// TwinCAT 3 PLC project CX747246
// ProgramVersion: 3.1.4024.0
// libraries:
//   CmpBitmapPool, * (System)
//   Tc2_Standard, * (Beckhoff Automation GmbH)
//   Tc2_SUPS, * (Beckhoff Automation GmbH)
//   Tc2_System, * (Beckhoff Automation GmbH)
//   Tc2_Utilities, * (Beckhoff Automation GmbH)
//   Tc3_EventLogger, * (Beckhoff Automation GmbH)
//   Tc3_Module, * (Beckhoff Automation GmbH)
//   VisuDialogs, * (System)
//   VisuElemEventTable, * (System)
//   VisuUserMgmt, * (System)
//   Visu Utils,3.5.12.0,System
//   VisuSymbols,3.5.10.0,System
// project tree:
//   DUTs/ StrFuncParoEnviar.TcDUT, Str_Config_ADS_to_PLC.TcDUT, Str_HistTablasMySQL.TcDUT
//   / GlobalTextList.TcGTLO, Lectura_PLCs_1.TcTTO, PlcTask.TcTTO, VISU_TASK.TcTTO
//   GVLs/ Fecha_PLC.TcGVL, Lectura_PLCs.TcGVL, RegistroLocalDataBase.TcGVL, Var_Com_CH4_MulDis.TcGVL
//   POUs/Events_Alarms/ Eventos_PLC.TcPOU, Events.TcPOU
//   POUs/FBs/ fbLectura_a_PLC.TcPOU, fb_Funciones_Paro.TcPOU, FuncGeneralesCortHum4.TcPOU, FuncGeneralesMult1.TcPOU, FuncGeneralesMult2.TcPOU, TempParoAcumulad.TcPOU
//   POUs/Funciones comunes/ Fecha_Hora_PLC.TcPOU, HMI.TcPOU, Utilidades.TcPOU
//   POUs/Lectura_a_PLC_Maestro/ Lectura_Maestro.TcPOU, MAIN_Orden_Lectura_PLCs.TcPOU
//   POUs/ MAIN.TcPOU
//   POUs/PRGs_Nodos/ FuncParoNodoMultidiscos.TcPOU, FuncParoNodoCorteH4Remote1.TcPOU
//   VISUs/ Ajustes_Multidiscos1.TcVIS, Ajustes_Multidiscos2.TcVIS, DiagnosticoFB.TcVIS, Home_CortH4.TcVIS, Home_Multidis1.TcVIS, Home_Multidis2.TcVIS, ImagePool.TcIPO (not stored), Modelo_Tabla_Ch4.TcVIS, Ajustes_CorteH4.TcVIS, Home_Sel_Maq.TcVIS, HistTablaTablas_Ch4.TcVIS, Modelo_Tabla_Md1.TcVIS, Modelo_Tabla_Md2.TcVIS, VisualizationManager.TcVMO (not stored), V_Emerg_Fin_Prod_Ch4.TcVIS, V_Emerg_Fin_Prod_Md2.TcVIS, V_Emerg_Fin_Prod_Md1.TcVIS
//   VISUs/IMAGENES/ Imagenes.TcIPO (not stored)
//   VISUs/Listas_Para_Desplegables/ FormatoTabla.TcTLO
// real-time tasks:
//   TASK PlcTask: cycle T#10ms, priority 20, ADS port 350
//   TASK VISU_TASK: cycle T#200000us, priority 30, ADS port 352
//   TASK Lectura_PLCs: cycle T#10ms, priority 1, ADS port 351
// I/O:
//   DEVICE Device 2 (EtherCAT), AmsNetId 5.116.114.70.3.1
//     Term 1 (EK1200) [EK1200-5000 EtherCAT Power supply (2A E-Bus)]
//       Term 2 (EL1859) [EL1859 8Ch. Dig. Input 24V, 3ms, 8Ch. Dig. Output 24V, 0.5A]
//       Term 3 (EK1110) [EK1110 EtherCAT extension]
//     Term 4 (EK1100) [EK1100 EtherCAT Coupler (2A E-Bus)]
//       Term 5 (EL1859) [EL1859 8Ch. Dig. Input 24V, 3ms, 8Ch. Dig. Output 24V, 0.5A]
//       Term 6 (EL9011) [EL9011 End Terminal]
// variable links:
//   CX747246/CX747246 Instance <-> Device 2 (EtherCAT)/Term 1 (EK1200)/Term 2 (EL1859)
//     PlcTask Inputs/MAIN.id0Local <-> Channel 1/Input
//     PlcTask Inputs/MAIN.id0Local @bit {1..7} <-> Channel {2..8}/Input  (7 links)
//     PlcTask Outputs/MAIN.od0Local @bit {1..7} <-> Channel {10..16}/Output  (7 links)
//     PlcTask Outputs/MAIN.od0Local <-> Channel 9/Output
//   CX747246/CX747246 Instance <-> Device 2 (EtherCAT)/Term 4 (EK1100)/Term 5 (EL1859)
//     PlcTask Inputs/MAIN.id0Remoto1 <-> Channel 1/Input
//     PlcTask Inputs/MAIN.id0Remoto1 @bit {1..7} <-> Channel {2..8}/Input  (7 links)
//     PlcTask Outputs/MAIN.od0Remoto1 @bit {1..7} <-> Channel {10..16}/Output  (7 links)
//     PlcTask Outputs/MAIN.od0Remoto1 <-> Channel 9/Output

CONFIGURATION CX747246
    RESOURCE PLC ON TwinCAT3
        TASK Lectura_PLCs_1(INTERVAL := T#10ms, PRIORITY := 1);
        TASK PlcTask(INTERVAL := T#10ms, PRIORITY := 20);
        TASK VISU_TASK(INTERVAL := T#200000us, PRIORITY := 30);
        PROGRAM MAIN_Orden_Lectura_PLCs WITH Lectura_PLCs_1 : MAIN_Orden_Lectura_PLCs;
        PROGRAM MAIN WITH PlcTask : MAIN;
        PROGRAM VisuElems_Visu_Prg WITH VISU_TASK : VisuElems.Visu_Prg;
        PROGRAM HMI WITH VISU_TASK : HMI;
    END_RESOURCE
END_CONFIGURATION

// ---- DUTs/StrFuncParoEnviar.TcDUT
TYPE StrFuncParoEnviar :
STRUCT
	Cont_Piezas:INT;//Numero de piezas actuales
	Min_Parado_Ftc:INT;//Minutos actuales parado
	t_Entr_Piez_Ante_Ftc:TIME;//Tiempo entre piezas tabla anterior
	t_Entre_Piez_Ftc:TIME;//Tiempo actual entre piezas
	H_InParo_Ftc:STRING;//Variable de la hora de inicio del paro tipo STRING
	H_FinParo_Ftc:STRING;//Hora Fin del paro
	S_Justi_Paro_Ftc:STRING;//Justificación del paro string
	Fotocelula:BOOL;//Fotocelula física
	MParo_Ftc:BOOL;//Marca de paro 
	M_SinParo_Ftc:BOOL;//Marca de sin paro activo
	tFiltro_up_Ftc:BOOL;//Q del temporizador Up filtro fotocelula 
	tFiltro_down_Ftc:BOOL;//Q del temporizador Down filtro fotocelula 	
END_STRUCT
END_TYPE

// ---- DUTs/Str_Config_ADS_to_PLC.TcDUT
TYPE Str_Config_ADS_to_PLC :
STRUCT
    NETID     : T_AmsNetId;
    PORT      : T_AmsPort;
    IDXGRP    : UDINT;
    IDXOFFS   : UDINT;
    LEN       : UDINT;
    DESTADDR  : PVOID;
    READ      : BOOL;
    TMOUT     : TIME := DEFAULT_ADS_TIMEOUT;
	
//Output
	BUSY    : BOOL;
    ERR     : BOOL;
    ERRID   : UDINT;
END_STRUCT
END_TYPE

// ---- DUTs/Str_HistTablasMySQL.TcDUT
TYPE Str_HistTablasMySQL :
STRUCT
	ID:INT;
	Fecha:STRING;
	Modelo:STRING;
	Formato:STRING;
	Espesor:STRING;
	Maquina :STRING;	
	Cont_Piezas:INT;//Numero de piezas actuales
	t_Entre_Piez_Ftc:TIME;//Tiempo actual entre piezas
	S_Justi_Paro_Ftc:STRING;//Justificación del paro string	
END_STRUCT
END_TYPE

// ---- GVLs/Fecha_PLC.TcGVL
{attribute 'qualified_only'}
VAR_GLOBAL
	fbGetLocalSystemTime:FB_LocalSystemTime; //Lee la hora local del PLC 
	Fecha_Segundos:DINT;
	StringDateTime:STRING;
	StringDateHourMin:STRING;
	StringDate:STRING;
	StringTime:STRING;
	StringHora:STRING;
	StringMinutos:STRING;
	StringSegundos:STRING;
	StringMes:STRING;
	StringDia:STRING;
	StringAno:STRING;
	
	//concatenaciones de strings
	Mes_Dia_Hora_Min_Real:STRING;
	//Tipo time para poder restar horas 
	Fecha_Entera_Dt:DT;	
	Fecha_Struct: Tc2_Utilities.TIMESTRUCT;
	Fecha_Time_PLC:TIME;
	
END_VAR

// ---- GVLs/Lectura_PLCs.TcGVL
{attribute 'qualified_only'}
VAR_GLOBAL
										//	Variables Lectura de PLC Maestro
									
//Las marcas a las que hace referencia del plc Maestro para las Bool van de la %MB46110 a %MB46210
	aMasterBoolCom:ARRAY[0..100] OF BOOL;
	
//Las marcas a las que hace referencia del plc Maestro para las string van de la %MW41300 a %MW42515   
	aMasterStringCom:ARRAY[0..14] OF STRING;
	
//Las marcas a las que hace rreferencia del plc Maestro para las Time van de la %MW47210 a %MW47414
	aMasterTimeCom:ARRAY[0..50]OF TIME;	
	
//Las marcas a las que hace referencia del plc Maestro para las Words van de la %MW45050 a %MW45090
	aMasterWordCom:ARRAY[0..40] OF WORD;	

END_VAR

// ---- GVLs/RegistroLocalDataBase.TcGVL
{attribute 'qualified_only'}
VAR_GLOBAL
	aValoresTurnosAnt: ARRAY [0..50] OF StrFuncParoEnviar;//Cada fin de turno se envía los valores de la ultima tabla que ha psado y se queda guardado en esta array para enseñarlo por el Scada
END_VAR
VAR_GLOBAL PERSISTENT
	//Array para el histórico de las tablas enviado a la base de datos
	 aHistoricStrTablasCH4: ARRAY[0..100]OF Str_HistTablasMySQL;
	 aHistoricStrTablasMD1: ARRAY[0..100]OF Str_HistTablasMySQL;
	 aHistoricStrTablasMD2: ARRAY[0..100]OF Str_HistTablasMySQL;
END_VAR

// ---- GVLs/Var_Com_CH4_MulDis.TcGVL
{attribute 'qualified_only'}
VAR_GLOBAL
	// Variables Escritura en PLC Maestro 
	aStringCom AT %MW2000: ARRAY[0..97] OF STRING;	//(1 string = 81 MW)
	aWordCom AT %MW10000: ARRAY[0..249] OF WORD;	//(1 Word = 1MW)
	aBoolCom AT %MB10250: ARRAY[0..499] OF BOOL;	//(1 Bool = 1MB)
	aTimeCom AT %MW10750: ARRAY[0..124] OF TIME;	//(1 Time = 4MW)
END_VAR

// ---- POUs/Lectura_a_PLC_Maestro/MAIN_Orden_Lectura_PLCs.TcPOU
PROGRAM MAIN_Orden_Lectura_PLCs
VAR
	bHabilitarLecturaDePLCs : BOOL := TRUE;
	bHabilitaLectura_Maestro : BOOL:=TRUE;
	State_Lectura_PLC: (READING_PLC_WAITING, READING_PLC_MAESTRO, FINISH_ALL_OK);
	tReadState_Entre_Lecturas_PLCs:ton:=(PT:=T#5MS);
END_VAR

// POU para ordenar la lectura de los distintos PLCs para que nunca lean a la vez 

CASE State_Lectura_PLC OF 

	READING_PLC_WAITING:tReadState_Entre_Lecturas_PLCs(IN:=FALSE);	

	READING_PLC_MAESTRO:	IF bHabilitaLectura_Maestro THEN
						tReadState_Entre_Lecturas_PLCs(IN:=TRUE);	
							IF tReadState_Entre_Lecturas_PLCs.Q THEN 
								tReadState_Entre_Lecturas_PLCs(IN:=FALSE);
								Lectura_Maestro();
								Lectura_Maestro.fbLectura_a_PLC_Maestro.SetStartReading();
							END_IF
							IF Lectura_Maestro.bNextBlockToRead_L4_Done THEN

								Lectura_Maestro.fbLectura_a_PLC_Maestro.SetFalseBlockReadDone();
								State_Lectura_PLC := FINISH_ALL_OK; //Cuando se añada un PLC cambiad el nombre.
							END_IF
						ELSE 
							State_Lectura_PLC := FINISH_ALL_OK; //Cuando se añada un PLC cambiad el nombre.
							Lectura_Maestro.fbLectura_a_PLC_Maestro.SetFalseBlockReadDone();
					END_IF
					
	FINISH_ALL_OK: tReadState_Entre_Lecturas_PLCs(IN:=FALSE);	
					State_Lectura_PLC := READING_PLC_Maestro;				

END_CASE



//Habilitar la lectura de los PLCs
IF bHabilitarLecturaDePLCs THEN 
	SetStartReadingPLCs();
	ELSE
		State_Lectura_PLC:=READING_PLC_WAITING;
END_IF

METHOD SetStartReadingPLCs : BOOL
VAR_INPUT
END_VAR
IF State_Lectura_PLC = READING_PLC_WAITING THEN 
	State_Lectura_PLC := READING_PLC_Maestro;
END_IF
END_METHOD

END_PROGRAM

// ---- POUs/Lectura_a_PLC_Maestro/Lectura_Maestro.TcPOU
PROGRAM Lectura_Maestro
VAR
	// >>>>>>>>>>>>>>>>>>>>>>>>>>>>>>>>>>>>>>>>   Estructuras de configuración con la comunicación desde y hacia el PLC Maestro <<<<<<<<<<<<<<<<<<<<<<<<<<<<<<<<<<<<<<<<<<<<<<<<<
	
	//Recordar que el IDXOFFS debe ser el doble de la posición a la que queréis acceder Ejemplo: para leer los strings a partir de la dirección MW100 Debéis poner 200 en exadecimal (C8)
	
	//Configuración de la lectura de las variables Bool, IDXGRP:=16#4020(Hace referencia a la lectura de M),IDXOFFS:=16#B41E(%MB46110 a %MB46210), LEN : 101 Longitud bools leidos,DESTADDR:= ADR(Lectura_PLCs.aMasterBoolCom) Ubicación del array donde se guarda la lectura
	Config_Read_ADS_Bools_Maestro:Str_Config_ADS_to_PLC:=(NETID:='192.168.10.71.1.1', PORT:=851, IDXGRP:=16#4020,IDXOFFS:=16#B41E,LEN:=101,DESTADDR:= ADR(Lectura_PLCs.aMasterBoolCom));
	
	//Configuración de la lectura de las variables String, IDXGRP:=16#4020(Hace referencia a la lectura de M),IDXOFFS:= 16#142A8(%MW41300 a %MW42515 ( 15 word)),Longitud de bytes a leer 1215 bytes = 15 strings que son 81words por cada string. ,DESTADDR:= ADR(Lectura_PLCs.aMasterStringCom) Ubicación del array donde se guarda la lectura
	Config_Read_ADS_Strings_Maestro:Str_Config_ADS_to_PLC:=(NETID:='192.168.10.71.1.1', PORT:=851, IDXGRP:=16#4020,IDXOFFS:=16#142A8,LEN:=1215,DESTADDR:= ADR(Lectura_PLCs.aMasterStringCom));
	
	//Configuración de la lectura de las variables Times, IDXGRP:=16#4020(Hace referencia a la lectura de M),IDXOFFS:=16#16F30 ( %MW47210 a %MW47414 (204 word),LEN:= 204 Longitud de bytes a leer bytes = 200words    51 componentes,DESTADDR:= ADR(Lectura_PLCs.aMasterTimeCom) Ubicación del array donde se guarda la lectura
	Config_Read_ADS_Times_Maestro:Str_Config_ADS_to_PLC:=(NETID:='192.168.10.71.1.1', PORT:=851, IDXGRP:=16#4020,IDXOFFS:=16#16F30,LEN:= 204,DESTADDR:= ADR(Lectura_PLCs.aMasterTimeCom));
	
	//Configuración de la lectura de las variables Words, IDXGRP:=16#4020(Hace referencia a la lectura de M),IDXOFFS:=16#15FF4 ( %MW45050 a %MW45090 (40 word),82;//Longitud de bytes a leer 80 bytes = 40words   ,DESTADDR:= ADR(Lectura_PLCs.aMasteWordCom) Ubicación del array donde se guarda la lectura
	Config_Read_ADS_Words_Maestro:Str_Config_ADS_to_PLC:=(NETID:='192.168.10.71.1.1', PORT:=851, IDXGRP:=16#4020,IDXOFFS:=16#15FF4,LEN:=82,DESTADDR:= ADR(Lectura_PLCs.aMasterWordCom));
	
	
	fbLectura_a_PLC_Maestro:fbLectura_a_PLC;
	

END_VAR
VAR_INPUT
	bNextBlockToRead_L4_Done:BOOL;
END_VAR

fbLectura_a_PLC_Maestro(
	Config_PLC_ADS_Bools:=Config_Read_ADS_Bools_Maestro,
	Config_PLC_ADS_Strings:=Config_Read_ADS_Strings_Maestro,
	Config_PLC_ADS_Times:=Config_Read_ADS_Times_Maestro,
	Config_PLC_ADS_Words:=Config_Read_ADS_Words_Maestro,
 	TimeReadStateEntreLecturas:=T#20MS,
	bHabilitadaLectura:=TRUE,
	);

END_PROGRAM

// ---- POUs/FBs/fbLectura_a_PLC.TcPOU
FUNCTION_BLOCK fbLectura_a_PLC
VAR_INPUT
	TimeReadStateEntreLecturas:TIME;
	//Estructuras para la configuración de la lectura de lsa ubicaciones de las variables y los tipos en el PLC 
	Config_PLC_ADS_Bools:Str_Config_ADS_to_PLC;
	Config_PLC_ADS_Strings:Str_Config_ADS_to_PLC;
	Config_PLC_ADS_Times:Str_Config_ADS_to_PLC;
	Config_PLC_ADS_Words:Str_Config_ADS_to_PLC;
	bHabilitadaLectura:BOOL;	
END_VAR 

VAR_OUTPUT
	AlarmaFalloComunicacion:BOOL;
END_VAR
VAR


	
	//Tiempos para el control de las lecturas de los diferentes tipos de variables
	tReadState_Entre_Lecturas:ton;
	eReadState : (EN_ESPERA,READING_BOOLS,READING_STRINGS,READING_TIMES,READING_WORDS,END_ALL_OK);
	//Bits de activación de lectura de las variables
	Execute_Read_Bools:BOOL;
	Execute_Read_Strings:BOOL;
	Execute_Read_Times:BOOL;
	Execute_Read_Words:BOOL;
	
	//Alarmas Errores en las lecturas al PLC 
	Err_fbLecturaBools: BOOL;
	Err_ID_fbLecturaBools: UDINT;
	Err_fbLecturaStrings: BOOL;
	Err_ID_fbLecturaStrings: UDINT;
	Err_fbLecturaTimes: BOOL;
	Err_ID_fbLecturaTimes: UDINT;
	Err_fbLecturaWords: BOOL;
	Err_ID_fbLecturaWords: UDINT;
	
	
	//Instancias de las funciones de lectura
	fbLecturaWords:        adsRead;	
	fbLecturaTimes:        adsRead;	
	fbLecturaStrings:      adsRead;
	fbLecturaBools:        adsRead;
	bBlock_Read_Done : BOOL;
		//Comprobaciones 
	Cont_Bool:INT;
	Cont_Str:INT;
	Cont_Word:INT;
	Cont_Time:INT;
	
	fptReadState_Entre_Lecturas:R_trig;

END_VAR
VAR PERSISTENT

END_VAR

tReadState_Entre_Lecturas(PT:=TimeReadStateEntreLecturas);
CASE eReadState OF 
	EN_ESPERA :   	tReadState_Entre_Lecturas(IN:=FALSE);

	READING_BOOLS : tReadState_Entre_Lecturas(IN:=TRUE);
					Read_Bools();
					IF tReadState_Entre_Lecturas.Q THEN
						tReadState_Entre_Lecturas(IN:=FALSE);
					    Cont_Bool:=Cont_Bool + 1;
						Execute_Read_Bools:=TRUE;
 						eReadState := READING_STRINGS;
					END_IF
	
	READING_STRINGS :tReadState_Entre_Lecturas(IN:=TRUE);
						Read_Strings();
					IF tReadState_Entre_Lecturas.Q THEN 
					    tReadState_Entre_Lecturas(IN:=FALSE);
						Execute_Read_Strings:=TRUE;
						Cont_Str:=Cont_Str + 1;	
						eReadState := READING_TIMES;
			
					END_IF
					
	READING_TIMES : tReadState_Entre_Lecturas(IN:=TRUE);
					Read_Times();
					IF tReadState_Entre_Lecturas.Q THEN 
						tReadState_Entre_Lecturas(IN:=FALSE);
						Execute_Read_Times:=TRUE;
						Cont_Time:=Cont_Time + 1;	
						eReadState := READING_WORDS;	
					END_IF
					
	READING_WORDS : tReadState_Entre_Lecturas(IN:=TRUE);
					Read_Words();
					IF tReadState_Entre_Lecturas.Q THEN 
						tReadState_Entre_Lecturas(IN:=FALSE);
						Execute_Read_Words:=TRUE;
						Cont_Word:=Cont_Word + 1;	
						eReadState := END_ALL_OK;	
									
					END_IF

	END_ALL_OK :// eReadState := READING_BOOLS;
				bBlock_Read_Done:=TRUE;
END_CASE

//En espera en caso de estar deshabilitado
IF NOT bHabilitadaLectura THEN
		eReadState:= EN_ESPERA;
END_IF
IF Err_fbLecturaBools OR Err_fbLecturaStrings OR Err_fbLecturaTimes OR Err_fbLecturaWords THEN 
	AlarmaFalloComunicacion:=TRUE;
	ELSE 
		AlarmaFalloComunicacion:=false;
END_IF

METHOD Read_Bools : BOOL
VAR_INPUT
END_VAR
fbLecturaBools.NETID:=  Config_PLC_ADS_Bools.NETID;//Lee del equipo remoto los Bool 
fbLecturaBools.PORT:=   Config_PLC_ADS_Bools.PORT;
fbLecturaBools.IDXGRP:= Config_PLC_ADS_Bools.IDXGRP;//Variables %M
fbLecturaBools.IDXOFFS:= Config_PLC_ADS_Bools.IDXOFFS;//Offset de la marca que empieza a leer
fbLecturaBools.LEN:= Config_PLC_ADS_Bools.LEN;//Longitud de bits a leer
fbLecturaBools.DESTADDR:= Config_PLC_ADS_Bools.DESTADDR;//Numero componentes
fbLecturaBools.READ:=     Execute_Read_Bools;//Bit de ejecutar la lectura 
fbLecturaBools();
Err_fbLecturaBools := fbLecturaBools.ERR;
Err_ID_fbLecturaBools := fbLecturaBools.ERRID;

Execute_Read_Bools := FALSE;
END_METHOD

METHOD Read_Strings : BOOL
VAR_INPUT
END_VAR
fbLecturaStrings.NETID:=  Config_PLC_ADS_Strings.NETID;//Lee del equipo remoto String
fbLecturaStrings.PORT:=   Config_PLC_ADS_Strings.PORT;
fbLecturaStrings.IDXGRP:= Config_PLC_ADS_Strings.IDXGRP;//Variables %M
fbLecturaStrings.IDXOFFS:= Config_PLC_ADS_Strings.IDXOFFS;//Offset 
fbLecturaStrings.LEN:= Config_PLC_ADS_Strings.LEN;//Longitud de bytes a leer 
fbLecturaStrings.DESTADDR:= Config_PLC_ADS_Strings.DESTADDR;//componentes
fbLecturaStrings.READ:=     Execute_Read_Strings;
fbLecturaStrings();
Err_fbLecturaStrings:= fbLecturaStrings.ERR;
Err_ID_fbLecturaStrings:= fbLecturaStrings.ERRID;


Execute_Read_Strings:=FALSE;
END_METHOD

METHOD Read_Times : BOOL
VAR_INPUT
END_VAR

fbLecturaTimes.NETID:=  Config_PLC_ADS_Times.NETID;//Lee del equipo remoto variables time
fbLecturaTimes.PORT:=   Config_PLC_ADS_Times.Port; //Puerto a leer
fbLecturaTimes.IDXGRP:= Config_PLC_ADS_Times.IDXGRP;//Variables %M
fbLecturaTimes.IDXOFFS:= Config_PLC_ADS_Times.IDXOFFS;//Offset 
fbLecturaTimes.LEN:= Config_PLC_ADS_Times.LEN;//Longitud de bytes a leer 
fbLecturaTimes.DESTADDR:= Config_PLC_ADS_Times.DESTADDR;// componentes
fbLecturaTimes.READ:=    Execute_Read_Times;
fbLecturaTimes();
Err_fbLecturaTimes:= fbLecturaTimes.ERR;
Err_ID_fbLecturaTimes:= fbLecturaTimes.ERRID;

Execute_Read_Times:=FALSE;
END_METHOD

METHOD Read_Words : BOOL
VAR_INPUT
END_VAR

fbLecturaWords.NETID:=  Config_PLC_ADS_Words.NETID;//Lee del equipo remoto variables words
fbLecturaWords.PORT:=   Config_PLC_ADS_Words.Port; //Puerto
fbLecturaWords.IDXGRP:= Config_PLC_ADS_Words.IDXGRP;//Variables %M
fbLecturaWords.IDXOFFS:= Config_PLC_ADS_Words.IDXOFFS;//Offset 
fbLecturaWords.LEN:= Config_PLC_ADS_Words.LEN;//Longitud de bytes a leer 
fbLecturaWords.DESTADDR:= Config_PLC_ADS_Words.DESTADDR;//Componentes
fbLecturaWords.READ:=  Execute_Read_Words ;
fbLecturaWords();
Err_fbLecturaWords:= fbLecturaWords.ERR;
Err_ID_fbLecturaWords:= fbLecturaWords.ERRID;

Execute_Read_Words:=FALSE;
END_METHOD

METHOD SetFalseBlockReadDone : BOOL
VAR_INPUT
END_VAR
	bBlock_Read_Done := FALSE;
	Execute_Read_Bools:= FALSE;
	Execute_Read_Strings:= FALSE;
	Execute_Read_Times:= FALSE;
	Execute_Read_Words:= FALSE;
END_METHOD

METHOD SetStartReading : BOOL
VAR_INPUT
	
END_VAR
IF eReadState = EN_ESPERA OR eReadState = END_ALL_OK THEN
	eReadState := READING_BOOLS;
END_IF
END_METHOD

END_FUNCTION_BLOCK

// ---- POUs/MAIN.TcPOU
PROGRAM MAIN
VAR
			// UPS variables persistentes
	fbUPS: FB_S_UPS_CX81xx;//Instancia de la UPS
	// Entradas
	id0Local   AT %I*: BYTE;
	id0Remoto1 AT %I*: BYTE;
	// Salidas
	od0Local   AT %Q*: BYTE;
	od0Remoto1 AT %Q*: BYTE;
	fbUtilidades: Utilidades;
END_VAR

fbUPS(iPLCPort:= 851,);
Fecha_Hora_PLC();
FuncParoNodoCorteH4Remote1();
FuncParoNodoMultidiscos();
Events();
fbUtilidades();

END_PROGRAM

// ---- POUs/Funciones comunes/Utilidades.TcPOU
FUNCTION_BLOCK Utilidades
VAR_INPUT
END_VAR
VAR_OUTPUT
END_VAR
VAR
sJustificaParoComun:STRING;
END_VAR

//Direccionamiento de variables para enviar 
Var_Com_CH4_MulDis.aStringCom[62] := Fecha_PLC.StringDateHourMin;

END_FUNCTION_BLOCK

// ---- POUs/Funciones comunes/Fecha_Hora_PLC.TcPOU
PROGRAM Fecha_Hora_PLC
VAR
END_VAR
VAR_TEMP
	HoraTemporal: STRING;
	
END_VAR

//Función para leer la fecha y hora del PLC 
Fecha_PLC.fbGetLocalSystemTime(
	sNetID:= , 
	bEnable:=TRUE , 
	dwCycle:=1 , 
	dwOpt:= , 
	tTimeout:= , 
	bValid=> , 
	systemTime=> , 
	tzID=> );
	
//Enviar la fecha y hora a una STRING
Fecha_PLC.StringDateTime:= SYSTEMTIME_TO_STRING(Fecha_PLC.fbGetLocalSystemTime.systemTime);

//Convertir a time la hora actual para poder realizar las restas entre fechas
Fecha_PLC.Fecha_Struct :=Fecha_PLC.fbGetLocalSystemTime.systemTime;
Fecha_PLC.Fecha_Entera_Dt:= SYSTEMTIME_TO_DT (Fecha_PLC.Fecha_Struct);
Fecha_PLC.Fecha_Time_PLC := DT_TO_TIME (Fecha_PLC.Fecha_Entera_Dt);


//Dividir en variables la fecha y hora STRING
Fecha_PLC.StringDate := MID(STR:= Fecha_PLC.StringDateTime, LEN:= 10, POS:= 1);
Fecha_PLC.StringDateHourMin := MID(STR:= Fecha_PLC.StringDateTime, LEN:= 19, POS:= 1);
Fecha_PLC.StringTime := MID(STR:= Fecha_PLC.StringDateTime, LEN:= 8, POS:= 12);
Fecha_PLC.StringAno := MID(STR:= Fecha_PLC.StringDateTime, LEN:= 4, POS:= 1);
Fecha_PLC.StringMes := MID(STR:= Fecha_PLC.StringDateTime, LEN:= 2, POS:= 6);
Fecha_PLC.StringDia := MID(STR:= Fecha_PLC.StringDateTime, LEN:= 2, POS:= 9);
Fecha_PLC.StringHora := MID(STR:= Fecha_PLC.StringDateTime, LEN:= 1, POS:= 12);
IF Fecha_PLC.StringHora = '0' THEN 
	Fecha_PLC.StringHora := MID(STR:= Fecha_PLC.StringDateTime, LEN:= 1, POS:= 13);
	ELSE 
		Fecha_PLC.StringHora := MID(STR:= Fecha_PLC.StringDateTime, LEN:= 2, POS:= 12);
END_IF
Fecha_PLC.StringMinutos := MID(STR:= Fecha_PLC.StringDateTime, LEN:= 2, POS:= 15);
Fecha_PLC.StringSegundos := MID(STR:= Fecha_PLC.StringDateTime, LEN:= 2, POS:= 18);

//Concatenacion de strings
	//Mes_Dia Hora:Minutos
	Fecha_PLC.Mes_Dia_Hora_Min_Real := concat(Fecha_PLC.StringDia,'_');
	Fecha_PLC.Mes_Dia_Hora_Min_Real:= concat(Fecha_PLC.Mes_Dia_Hora_Min_Real,Fecha_PLC.StringMes); 
	Fecha_PLC.Mes_Dia_Hora_Min_Real:= concat(Fecha_PLC.Mes_Dia_Hora_Min_Real,'  ');
	Fecha_PLC.Mes_Dia_Hora_Min_Real:= concat(Fecha_PLC.Mes_Dia_Hora_Min_Real,Fecha_PLC.StringHora);
	Fecha_PLC.Mes_Dia_Hora_Min_Real:= concat(Fecha_PLC.Mes_Dia_Hora_Min_Real,':');
	Fecha_PLC.Mes_Dia_Hora_Min_Real:= concat(Fecha_PLC.Mes_Dia_Hora_Min_Real,Fecha_PLC.StringMinutos);

END_PROGRAM

// ---- POUs/PRGs_Nodos/FuncParoNodoCorteH4Remote1.TcPOU
PROGRAM FuncParoNodoCorteH4Remote1
VAR
	Funci_CortHum4:fb_Funciones_Paro;
	FunGeneCortHum4: FuncGeneralesCortHum4;
	//Entradas Corte húmedo 4
	Ftc_CortHum4: BOOL;	
	ForzadoFtcCortHum4:BOOL;	
	Consenso_CortHum4: BOOL;
	//Entradas fotocelula 2 libre
	Ftc2_Libre: BOOL;
	ForzadoFtc2_Libre: BOOL;
	Consenso_Ftc2_Libre: BOOL;
	//Entradas fotocelula 3 libre
	Ftc3_Libre: BOOL;
	ForzadoFtc3_Libre: BOOL;
	Consenso_Ftc3_Libre: BOOL;
	//Entradas fotocelula 4 libre
	Ftc4_Libre: BOOL;
	ForzadoFtc4_Libre: BOOL;
	Consenso_Ftc4_Libre: BOOL;
	
//	Estructuras de las variables a enviar  
	CortHum4StrFuncParoEnviar:StrFuncParoEnviar;
	Ftc2StrFuncParoEnviar:StrFuncParoEnviar;	
	Ftc3StrFuncParoEnviar:StrFuncParoEnviar;
	Ftc4StrFuncParoEnviar:StrFuncParoEnviar;
	

END_VAR
VAR_INPUT
	sFormatoEleccionTabla:STRING;
	sModeloEleccionTabla:STRING;
	sEspesorEleccionTabla:STRING;
END_VAR
VAR RETAIN
END_VAR
VAR PERSISTENT 
	HMI_Tiempo_Offset_MParo:INT:=5;
	HMI_TiempoFiltradoFotocel:TIME:=T#2S;
// Modelo de la tabla y fecha cambio de modelo
	sModeloActualTabla:STRING;
	sFormatoActualTabla:STRING;
	sEspesorActualTabla:STRING;
	sFechaInicModeloTab:STRING;


END_VAR

//Funciones de paro para cada zona(Fotocelula)

//>>>>>>>>>>>>>>>>>>>>>>>>>>>>>>>>>>>>>>>>>>>>>         	Corte húmedo 4         <<<<<<<<<<<<<<<<<<<<<<<<<<<<<<<<<<<<<<<<<<<<<<<<<<<<<<<<<<
Funci_CortHum4(Fotocelula:=Ftc_CortHum4 OR ForzadoFtcCortHum4, 
					Tiempo_Offset_MParo:=HMI_Tiempo_Offset_MParo, 
					TiempoFiltradoFotocel:=HMI_TiempoFiltradoFotocel,
					_StrFuncParoEnviar => CortHum4StrFuncParoEnviar );
					
						
						
Direccionamiento_variables_com();
LinkadoEntradas();
FunGeneCortHum4(s_ModeloActualTabla => sModeloActualTabla,s_ModeloEleccionTabla => sModeloEleccionTabla,s_FechaInicModeloTab=>sFechaInicModeloTab,s_FormatoActualTabla=>sFormatoActualTabla,s_FormatoEleccionTabla=>sFormatoEleccionTabla,s_EspesorActualTabla=>sEspesorActualTabla,s_EspesorEleccionTabla=>sEspesorEleccionTabla);

ACTION Direccionamiento_variables_com:
// Direccionamiento de las variables a la marca que les corresponde donde despés se leeran desde el plc maestro



//								>>>>>>>>>>>>>>>>>>>>>>>>>>>>      WORDS    <<<<<<<<<<<<<<<<<<<<<<<<<<<<<<<<

	Var_Com_CH4_MulDis.aWordCom[50]:= INT_TO_WORD (CortHum4StrFuncParoEnviar.Cont_Piezas);	    //Contadores de cada fotocelula 
	Var_Com_CH4_MulDis.aWordCom[51]:= INT_TO_WORD (Ftc2StrFuncParoEnviar.Cont_Piezas);		//Contadores de cada fotocelula 
	Var_Com_CH4_MulDis.aWordCom[52]:= INT_TO_WORD (Ftc3StrFuncParoEnviar.Cont_Piezas);		//Contadores de cada fotocelula 
	Var_Com_CH4_MulDis.aWordCom[53]:= INT_TO_WORD (Ftc4StrFuncParoEnviar.Cont_Piezas);		//Contadores de cada fotocelula 
	Var_Com_CH4_MulDis.aWordCom[54]:= INT_TO_WORD (CortHum4StrFuncParoEnviar.Min_Parado_Ftc);			//Minutos actuales parado
	Var_Com_CH4_MulDis.aWordCom[55]:= INT_TO_WORD (Ftc2StrFuncParoEnviar.Min_Parado_Ftc);			//Minutos actuales parado
	Var_Com_CH4_MulDis.aWordCom[56]:= INT_TO_WORD (Ftc3StrFuncParoEnviar.Min_Parado_Ftc);			//Minutos actuales parado
	Var_Com_CH4_MulDis.aWordCom[57]:= INT_TO_WORD (Ftc4StrFuncParoEnviar.Min_Parado_Ftc);			//Minutos actuales parado
	
	
	
//                           	>>>>>>>>>>>>>>>>>>>>>>>>>>>>      TIME   <<<<<<<<<<<<<<<<<<<<<<<<<<<<<<<<
	
	
	Var_Com_CH4_MulDis.aTimeCom[25]:=  CortHum4StrFuncParoEnviar.t_Entre_Piez_Ftc; 			//Tiempo entre piezas
	Var_Com_CH4_MulDis.aTimeCom[26]:=  Ftc2StrFuncParoEnviar.t_Entre_Piez_Ftc;			//Tiempo entre piezas
	Var_Com_CH4_MulDis.aTimeCom[27]:= Ftc3StrFuncParoEnviar.t_Entre_Piez_Ftc;				//Tiempo entre piezas
	Var_Com_CH4_MulDis.aTimeCom[28]:= Ftc4StrFuncParoEnviar.t_Entre_Piez_Ftc;				//Tiempo entre piezas
	Var_Com_CH4_MulDis.aTimeCom[29]:= CortHum4StrFuncParoEnviar.t_Entr_Piez_Ante_Ftc; 		//Tiempo entre piezas anterior
	Var_Com_CH4_MulDis.aTimeCom[30]:= Ftc2StrFuncParoEnviar.t_Entr_Piez_Ante_Ftc; 		//Tiempo entre piezas anterior
	Var_Com_CH4_MulDis.aTimeCom[31]:= Ftc3StrFuncParoEnviar.t_Entr_Piez_Ante_Ftc; 		//Tiempo entre piezas anterior
	Var_Com_CH4_MulDis.aTimeCom[32]:= Ftc4StrFuncParoEnviar.t_Entr_Piez_Ante_Ftc; 		//Tiempo entre piezas anterior
	
	
	
	
//                           	>>>>>>>>>>>>>>>>>>>>>>>>>>>>      STRING  <<<<<<<<<<<<<<<<<<<<<<<<<<<<<<<<
    Var_Com_CH4_MulDis.aStringCom[20] := CortHum4StrFuncParoEnviar.H_InParo_Ftc;         //Hora inicio paro 
	Var_Com_CH4_MulDis.aStringCom[21] := Ftc2StrFuncParoEnviar.H_InParo_Ftc;         //Hora inicio paro 
	Var_Com_CH4_MulDis.aStringCom[22] := Ftc3StrFuncParoEnviar.H_InParo_Ftc;         //Hora inicio paro 
	Var_Com_CH4_MulDis.aStringCom[23] := Ftc4StrFuncParoEnviar.H_InParo_Ftc;         //Hora inicio paro 
	Var_Com_CH4_MulDis.aStringCom[24] := CortHum4StrFuncParoEnviar.H_FinParo_Ftc;        //Hora Fin paro 
	Var_Com_CH4_MulDis.aStringCom[25] := Ftc2StrFuncParoEnviar.H_FinParo_Ftc;        //Hora Fin paro 
	Var_Com_CH4_MulDis.aStringCom[26] := Ftc3StrFuncParoEnviar.H_FinParo_Ftc;        //Hora Fin paro 
	Var_Com_CH4_MulDis.aStringCom[27] := Ftc4StrFuncParoEnviar.H_FinParo_Ftc;        //Hora Fin paro 
	Var_Com_CH4_MulDis.aStringCom[28] := CortHum4StrFuncParoEnviar.S_Justi_Paro_Ftc;		//Justificación del paro
	Var_Com_CH4_MulDis.aStringCom[29] := Ftc2StrFuncParoEnviar.S_Justi_Paro_Ftc;		//Justificación del paro
	Var_Com_CH4_MulDis.aStringCom[30] := Ftc3StrFuncParoEnviar.S_Justi_Paro_Ftc;		//Justificación del paro
	Var_Com_CH4_MulDis.aStringCom[31] := Ftc4StrFuncParoEnviar.S_Justi_Paro_Ftc;		//Justificación del paro
	
	
//                           	>>>>>>>>>>>>>>>>>>>>>>>>>>>>      Bool  <<<<<<<<<<<<<<<<<<<<<<<<<<<<<<<<	

	Var_Com_CH4_MulDis.aBoolCom[99] := CortHum4StrFuncParoEnviar.Fotocelula;						//Fotocelula Real
	Var_Com_CH4_MulDis.aBoolCom[100] := Ftc2StrFuncParoEnviar.Fotocelula;						//Fotocelula Real
	Var_Com_CH4_MulDis.aBoolCom[101] := Ftc3StrFuncParoEnviar.Fotocelula;						//Fotocelula Real
	Var_Com_CH4_MulDis.aBoolCom[102] := Ftc4StrFuncParoEnviar.Fotocelula;						//Fotocelula Real
	Var_Com_CH4_MulDis.aBoolCom[103] := CortHum4StrFuncParoEnviar.MParo_Ftc;				//Marca de paro 
	Var_Com_CH4_MulDis.aBoolCom[104] := Ftc2StrFuncParoEnviar.MParo_Ftc;				//Marca de paro 
	Var_Com_CH4_MulDis.aBoolCom[105] := Ftc3StrFuncParoEnviar.MParo_Ftc;				//Marca de paro 
	Var_Com_CH4_MulDis.aBoolCom[106] := Ftc4StrFuncParoEnviar.MParo_Ftc;				//Marca de paro 
	Var_Com_CH4_MulDis.aBoolCom[107] := CortHum4StrFuncParoEnviar.M_SinParo_Ftc;			//Marca de sin paro activo
	Var_Com_CH4_MulDis.aBoolCom[108] := Ftc2StrFuncParoEnviar.M_SinParo_Ftc;			//Marca de sin paro activo
	Var_Com_CH4_MulDis.aBoolCom[109] := Ftc3StrFuncParoEnviar.M_SinParo_Ftc;			//Marca de sin paro activo
	Var_Com_CH4_MulDis.aBoolCom[110] := Ftc4StrFuncParoEnviar.M_SinParo_Ftc;			//Marca de sin paro activo
	Var_Com_CH4_MulDis.aBoolCom[111] := CortHum4StrFuncParoEnviar.tFiltro_up_Ftc;			//Q Temp Up Filtro Fotocelulas
	Var_Com_CH4_MulDis.aBoolCom[112] := Ftc2StrFuncParoEnviar.tFiltro_up_Ftc;			//Q Temp Up Filtro Fotocelulas
	Var_Com_CH4_MulDis.aBoolCom[113] := Ftc3StrFuncParoEnviar.tFiltro_up_Ftc;			//Q Temp Up Filtro Fotocelulas
	Var_Com_CH4_MulDis.aBoolCom[114] := Ftc4StrFuncParoEnviar.tFiltro_up_Ftc;			//Q Temp Up Filtro Fotocelulas
	Var_Com_CH4_MulDis.aBoolCom[115] := CortHum4StrFuncParoEnviar.tFiltro_down_Ftc;		//Q Temp Down Filtro Fotocelulas
	Var_Com_CH4_MulDis.aBoolCom[116] := Ftc2StrFuncParoEnviar.tFiltro_down_Ftc;		//Q Temp Down Filtro Fotocelulas
	Var_Com_CH4_MulDis.aBoolCom[117] := Ftc3StrFuncParoEnviar.tFiltro_down_Ftc;		//Q Temp Down Filtro Fotocelulas
	Var_Com_CH4_MulDis.aBoolCom[118] := Ftc4StrFuncParoEnviar.tFiltro_down_Ftc;		//Q Temp Down Filtro Fotocelulas
END_ACTION

ACTION LinkadoEntradas:
// Linkado entradas

Ftc_CortHum4:=      main.id0Remoto1.0;
Consenso_CortHum4:= TRUE;//main.id0Remoto1.1;


Ftc2_Libre:=      main.id0Remoto1.2;
Consenso_Ftc3_Libre:= TRUE;// main.id0Remoto1.3;


Ftc3_Libre:=      main.id0Remoto1.4;
Consenso_Ftc3_Libre:= TRUE;// main.id0Remoto1.5;


Ftc4_Libre:=      main.id0Remoto1.6;
Consenso_Ftc4_Libre:= TRUE;// main.id0Remoto1.7;
END_ACTION

END_PROGRAM

// ---- POUs/FBs/fb_Funciones_Paro.TcPOU
FUNCTION_BLOCK fb_Funciones_Paro
VAR_INPUT
	Fotocelula: BOOL;
	Tiempo_Offset_MParo:INT;//Tiempo a partir del cual empieza a contar como paro
	TiempoFiltradoFotocel:TIME;
	Pul_Reset_Cnt_Piez : BOOL;
	S_Justi_Paro_Ftc:STRING;//Justificación del paro	
END_VAR
VAR_OUTPUT	
	tFiltro_up_Ftc:ton;//Temporizador de filtro parpadeos Up	
	tFiltro_down_Ftc:ton;//Temporizador de filtro parpadeos Down	
	MParo_Ftc:BOOL;//Marca de bit de linea parada en este momento	
	M_SinParo_Ftc:BOOL;//Marca de la linea sin paro (producción constante)	 
	H_FinParo_Ftc:STRING;//Variable de la hora de fin del paro	
	t_DetUp_Pieza:TIMESTRUCT;//Fecha detección positiva de pieza para tiempo entre piezas
	tH_FinParo_Ftc:STRING;//Variable de la hora de fin del paro tipo time	
	Min_Parado_Ftc:INT;//Minutos actuales parado	
	t_Entre_Piez_Ftc:TIME;//Minutos entre piezas 	
	M_Delay_Esc_Ftc:BOOL;//Delay escritura 	
	Delay_Esc_Ftc:ton;// tiempo Delay escritura 
	_StrFuncParoEnviar:StrFuncParoEnviar;
	t_Paro_Acumulado_Diario:TIME;
	t_Paro_Acumulado_Turno:TIME;
	t_Paro_Acumulado_Modelo:TIME;	
END_VAR
VAR RETAIN
	Cont_Piezas_Ftc:INT;	//Contador de piezas 				
	t_Entr_Piez_Ante_Ftc:TIME;//Minutos entre piezas tabla anterior 		
	tH_InParo_Ftc:STRING;//Variable de la hora de inicio del paro tipo STRING 
	t_InParo_Ftc_Entera:STRING;
	t_InParo_Ftc_Ent_Syst:TIMESTRUCT;	 
	H_InParo_Ftc:STRING;//Variable de la hora de inicio del paro
	
END_VAR
VAR
	i:INT;
	Temporizador1min:ton;
	FlancoUpFtc:R_TRIG;
	FlancoDoFtc:R_TRIG;
	FlancoFiltUpFtc:R_TRIG;
	FlancoFiltDoFtc:R_TRIG;
	tonTempON:ton;
	tonTempOFF:ton;
	tHoraReal:TIME;
	tHora:TIME;
	sHora: STRING(255);
	ResetContPiez:BOOL;
	s_Entr_Piez_Ante_Ftc:TIME;
	S_Entre_Piez_Ftc:TIME;
	fbTiempParoAcumTurno:TempParoAcumulad;
	fbTiempParoAcumDiario:TempParoAcumulad;
	fbTiempParoAcumModelo:TempParoAcumulad;
	Cont:INT;
	//Comprobaciones de los retardos de envio de frase a mysql a traves del maestro 
	TonAscendente:ton;
	Tiempo_Sumando:TIME:=T#3S;
	Tiempo_A_Sumar:TIME:=T#1.25S;
	ContandoComprobador:BOOL;
	bCompFuncEnvDataBase:BIT;
	TonOff:TON;
END_VAR


	//Llamada a los temporizadores Declaración de tiempos
		tFiltro_up_Ftc(PT:=TiempoFiltradoFotocel); 
		tFiltro_down_Ftc(PT:=TiempoFiltradoFotocel);
		Delay_Esc_Ftc(PT:=T#2S);//El delay funciona bien a T#2s
		
	// Temporizador para empezar a detectar pieza en paro (filtro de parpadeos) Up
	IF 	Fotocelula OR NOT tFiltro_down_Ftc.Q or ContandoComprobador THEN 
		tFiltro_up_Ftc.IN:=TRUE;
		ELSE
			 tFiltro_up_Ftc.IN:=FALSE;
	END_IF
	
	// Temporizador para empezar a detectar pieza en paro (filtro de parpadeos) Up
	IF 	NOT Fotocelula THEN 
		tFiltro_down_Ftc.IN:=TRUE;
		ELSE
			 tFiltro_down_Ftc.IN:=FALSE;
	END_IF

	//Tiempo real parado en minutos
	IF Temporizador1min.Q THEN 
		Min_Parado_Ftc:=Min_Parado_Ftc +1;		
	END_IF
	


//Crea flancos de subida cada vez que el temporizador de cada fotocelula se activa 
		//Flanco filtro Up ftc
		FlancoFiltUpFtc(CLK:=tFiltro_up_Ftc.Q);
		//Flanco filtro Down ftc
		FlancoFiltDoFtc(CLK:=tFiltro_down_Ftc.Q);	
		
//BIT Delay para Restar la hora inicio paro a la hora actual para sacar tiempo entre piezas(Dar tiempo a que el otro plc lea el valor de la variable antes del reset)
	IF FlancoFiltUpFtc.Q THEN
		 M_Delay_Esc_Ftc:= TRUE;			
	END_IF
	//Temporizador de retardo reset inicio del paro
	 	Delay_Esc_Ftc(IN:=M_Delay_Esc_Ftc);
	//Inserta en fecha inicio paro la hora actual y reset de valores
	IF Delay_Esc_Ftc.Q THEN
		Fecha_Inicio_Paro();
		Reset_Justif_Paro();		
		Min_Parado_Ftc:= 0;
		M_Delay_Esc_Ftc:= FALSE;
	END_IF
	
//Contador Piezas
  IF FlancoFiltUpFtc.Q THEN 
	  Cont_Piezas_Ftc:=Cont_Piezas_Ftc+1;
	  Resta_Tiempo_Entre_Piezas();
	  Fecha_Detec_Up_Pieza();
  END_IF
  
//Reset contador de las piezas
IF ResetContPiez THEN 
Reset_cnt_piez(Pul_Reset:=TRUE);  
  END_IF 
  
  
 //Instanciar todos los metodos que tengan que estar corriendo todo el tiempo y la dirección de sus entradas
Reset_cnt_piez(Pul_Reset:=Pul_Reset_Cnt_Piez);

//si el paro excede de el tiempo de la variable offset empieza a contar como paro y resetea marca sin paro 
Mparo_SinParo();
Temporizador1min(IN:=NOT Temporizador1min.Q , PT:= T#60S, Q=> , ET=> );
// Enviar constantemente la Fecha a Hora fin de paro 
Fin_Paro();
// Temporizadores acumulativos del paro, Turno, Diario, Modelo nuevo
TiempoParoAcumulado();
//Estructura de variables que luego de las cuales el PLC maestro leerá toda la información del paro
aStrFuncParEnviar();
IF  bCompFuncEnvDataBase THEN 
CompEnvContDataBase();
ELSE 
ContandoComprobador:=FALSE;	
END_IF

ACTION aStrFuncParEnviar:
_StrFuncParoEnviar.Cont_Piezas:=Cont_Piezas_Ftc;
_StrFuncParoEnviar.Fotocelula:=Fotocelula;
_StrFuncParoEnviar.H_FinParo_Ftc:=H_FinParo_Ftc;
_StrFuncParoEnviar.H_InParo_Ftc:=H_InParo_Ftc;
_StrFuncParoEnviar.M_SinParo_Ftc:= M_SinParo_Ftc;
_StrFuncParoEnviar.Min_Parado_Ftc:= Min_Parado_Ftc;
_StrFuncParoEnviar.MParo_Ftc:= MParo_Ftc;
_StrFuncParoEnviar.S_Justi_Paro_Ftc:=S_Justi_Paro_Ftc;
_StrFuncParoEnviar.t_Entr_Piez_Ante_Ftc:=t_Entr_Piez_Ante_Ftc;
_StrFuncParoEnviar.t_Entre_Piez_Ftc:=t_Entre_Piez_Ftc;
_StrFuncParoEnviar.tFiltro_down_Ftc:= tFiltro_down_Ftc.Q;
_StrFuncParoEnviar.tFiltro_up_Ftc:= tFiltro_up_Ftc.Q;
END_ACTION

METHOD CompEnvContDataBase : BOOL
VAR_INPUT
END_VAR
VAR 

END_VAR
//Está funcion está hecha para comprobar si los tiempos de retardo para la lectura a plc desde el plc esclavo al plc maestro junto los los retardos que tenga el maestro funcionan bien
//Cada cierto tiempo se va a incrementar en 10ms el temporizador , que será el encargado de forzar la fotocélula para enviar StrFuncParoEnviar.
TonAscendente(IN:=ContandoComprobador,PT:=Tiempo_Sumando);
TonOff(In:=NOT ContandoComprobador,Pt:=T#2S);
//ContandoComprobador:=TRUE;
IF TonAscendente.Q THEN 	
	Tiempo_Sumando:=Tiempo_Sumando + Tiempo_A_Sumar; 
	ContandoComprobador:=FALSE;
END_IF
IF Tiempo_Sumando > T#15S THEN
	Tiempo_Sumando:=T#1.25S;
END_IF
IF TonOff.Q THEN 
	ContandoComprobador:=TRUE;
END_IF
END_METHOD

METHOD Fecha_Detec_Up_Pieza : BOOL
VAR_INPUT
END_VAR
t_DetUp_Pieza:= Fecha_PLC.Fecha_Struct;
END_METHOD

METHOD Fecha_Inicio_Paro
VAR_INPUT
END_VAR
VAR 

END_VAR

//Envío la fecha entera de inicio paro en formato string  
t_InParo_Ftc_Entera:=Fecha_PLC.StringDateTime;
t_InParo_Ftc_Ent_Syst:= Fecha_PLC.Fecha_Struct ;
//Envío la fecha reducida de inicio paro en formato string para poder verla en HMI 
tH_InParo_Ftc:= Fecha_PLC.Mes_Dia_Hora_Min_Real;
H_InParo_Ftc:= Fecha_PLC.Mes_Dia_Hora_Min_Real;
END_METHOD

METHOD Fin_Paro : BOOL
VAR_INPUT
END_VAR

//Envío de la fecha actual completa para luego enviar a la base de datos 
tH_FinParo_Ftc:= Fecha_PLC.Mes_Dia_Hora_Min_Real;
//Envío de la fecha actual reducida para mostrarlo en el hmi del maestro
H_FinParo_Ftc:= Fecha_PLC.Mes_Dia_Hora_Min_Real;
END_METHOD

METHOD Fin_Produccion
VAR_INPUT
END_VAR

VAR
	H: INT;
END_VAR

//Se le llama desde un metodo de Datos comunes 
// Reset de los contadores
Cont_Piezas_Ftc:=0;
fbTiempParoAcumModelo.ResetContador();
END_METHOD

METHOD Mparo_SinParo : BOOL
VAR_INPUT
END_VAR
IF Tiempo_Offset_MParo <= Min_Parado_Ftc THEN
		MParo_Ftc:=TRUE;
		M_SinParo_Ftc:=FALSE;	
	ELSE 
		MParo_Ftc:=FALSE;
		M_SinParo_Ftc:=TRUE;	
END_IF
END_METHOD

METHOD Reset_cnt_piez : BOOL
VAR_INPUT
		Pul_Reset:BOOL;
END_VAR
VAR 

END_VAR
IF Pul_Reset THEN 
	Cont_Piezas_Ftc:=0;
	Cont:=Cont+1;
END_IF
END_METHOD

METHOD Reset_Justif_Paro : BOOL
VAR_INPUT
END_VAR
S_Justi_Paro_Ftc:='.';
END_METHOD

METHOD Resta_Tiempo_Entre_Piezas
VAR_INPUT 
END_VAR

VAR
	Dt_InParo_Entera:DATE_AND_TIME;
	Time_InParo_Entera:TIME;
	t_InParo_Ftc_Entera_Temp: TIMESTRUCT;
END_VAR
//Esta funcion al notar flanco positivo o negativo de la fotocelula 
//coge la Fecha actual en tipo time y la resta a la Hora inicio paro para sacar cuanto tiempo ha transcurrido entre piezas 
//No funciona bien si haces el cambio de string a Dt hay que hacerlo desde systemtime to Dt 

//Envío el tiempo entre tablas de la anterior a la variable que le toca 
t_Entr_Piez_Ante_Ftc:= t_Entre_Piez_Ftc;


//La hora de inicio paro entera la pasamos a una variable del metodo para poder trabajar con ella sin modificar la de la FB
t_InParo_Ftc_Entera_Temp := t_DetUp_Pieza;
//Convertir la fecha entera inicio de string a dt y después a time 
Dt_InParo_Entera:= SYSTEMTIME_TO_DT(t_InParo_Ftc_Entera_Temp);
Time_InParo_Entera:= DT_TO_TIME(Dt_InParo_Entera);

// Resta de la fecha de inicio entera Time menos fecha actual entera time
t_Entre_Piez_Ftc:= Fecha_PLC.Fecha_Time_PLC - Time_InParo_Entera ;
//t_Entre_Piez_Ftc:= Delete(t_Entre_Piez_Ftc,LEN:=2,POS:=1);
END_METHOD

METHOD TiempoParoAcumulado : BOOL
VAR_INPUT
END_VAR
VAR

END_VAR

//<<<<<<<<<<<<<<<<<<<<<<<<<<<<<<<< Reset contadores según tiempos >>>>>>>>>>>>>>>>>>>>>>>>>>>>>>>

//Diario 
IF Fecha_PLC.Fecha_Struct.wHour = 0 AND Fecha_PLC.Fecha_Struct.wMinute = 0 AND Fecha_PLC.Fecha_Struct.wSecond = 0 THEN 
	fbTiempParoAcumDiario.ResetContador();
END_IF

//Turno  
IF (Fecha_PLC.Fecha_Struct.wHour = 6 AND Fecha_PLC.Fecha_Struct.wMinute = 0 AND Fecha_PLC.Fecha_Struct.wSecond = 0)
 OR (Fecha_PLC.Fecha_Struct.wHour = 14 AND Fecha_PLC.Fecha_Struct.wMinute = 0 AND Fecha_PLC.Fecha_Struct.wSecond = 0)
 OR (Fecha_PLC.Fecha_Struct.wHour = 22 AND Fecha_PLC.Fecha_Struct.wMinute = 0 AND Fecha_PLC.Fecha_Struct.wSecond = 0)   
THEN 
	fbTiempParoAcumTurno.ResetContador();
END_IF

//Por modelo se reliza en el method Fin_Produccion


// Llamadas a los fb de los contadores acumulativos 
fbTiempParoAcumDiario(EnableCount:=tFiltro_up_Ftc.Q,
					  ParoActivo:=MParo_Ftc,
					  DateAndTimeActual:=Fecha_PLC.Fecha_Entera_Dt,
					  t_Acumulado=>t_Paro_Acumulado_Diario);
fbTiempParoAcumTurno(EnableCount:=tFiltro_up_Ftc.Q,
					  ParoActivo:=MParo_Ftc,
					  DateAndTimeActual:=Fecha_PLC.Fecha_Entera_Dt,
					  t_Acumulado=>t_Paro_Acumulado_Turno);
fbTiempParoAcumModelo(EnableCount:=tFiltro_up_Ftc.Q,
					  ParoActivo:=MParo_Ftc,
					  DateAndTimeActual:=Fecha_PLC.Fecha_Entera_Dt,
					  t_Acumulado=>t_Paro_Acumulado_Modelo);
END_METHOD

END_FUNCTION_BLOCK

// ---- POUs/FBs/TempParoAcumulad.TcPOU
FUNCTION_BLOCK TempParoAcumulad
VAR_INPUT
	EnableCount:BOOL;
	ParoActivo:BOOL;

	DateAndTimeActual:DATE_AND_TIME;
	P_resetCont:BOOL;
	
END_VAR
VAR_OUTPUT
	t_Acumulado:TIME;
END_VAR
VAR
	FlancoUp_Enable:r_trig;
	FlancoDo_Enable:f_trig;
	t_InicioSuma:TIME;
	t_FinSuma:TIME;
END_VAR

FlancoUp_Enable(CLK:=EnableCount);
FlancoDo_Enable(CLK:=EnableCount);

IF FlancoUp_Enable.Q THEN 
	InicioHoraCont();
END_IF
IF FlancoDo_Enable.Q AND ParoActivo THEN  
	FinHoraCont();
END_IF
IF P_resetCont THEN 
	ResetContador();
	P_resetCont:=FALSE;
END_IF

METHOD FinHoraCont : BOOL
VAR_INPUT
END_VAR
t_FinSuma := DT_TO_TIME(DateAndTimeActual);
t_Acumulado:= t_Acumulado + (t_FinSuma-t_InicioSuma);
END_METHOD

METHOD InicioHoraCont : BOOL
VAR_INPUT
END_VAR
t_InicioSuma := DT_TO_TIME(DateAndTimeActual) ;
END_METHOD

METHOD ResetContador : BOOL
VAR_INPUT
END_VAR
InicioHoraCont();
t_Acumulado:=T#0S;
END_METHOD

END_FUNCTION_BLOCK

// ---- POUs/FBs/FuncGeneralesCortHum4.TcPOU
FUNCTION_BLOCK FuncGeneralesCortHum4
VAR_INPUT
IndexListFormatoTabla:INT;
END_VAR
VAR_OUTPUT
	//Modelo dividido en strings para DataBase
	s_ModeloActualTabla:STRING;
	s_FormatoActualTabla:STRING;
	s_EspesorActualTabla:STRING;
	s_ModeloEleccionTabla:STRING;
	s_FormatoEleccionTabla:STRING;
	s_EspesorEleccionTabla:STRING;
	//Comunes
	s_JustificaParoComun:STRING;
	s_FechaInicModeloTab:STRING;
END_VAR
VAR
	Reset_Fin_Prod:BOOL;
	P_FinProduccion:BOOL;
	P_EscribirModelo:BOOL;
	pul_Justif_Paro:BOOL;
	EscribeHistoricTablas:BOOL;
	FlancFiltUpFtcEscHistTab:R_TRIG;
	Cont1:INT;
	Cont2:INT;
	Cont3:INT;
	Cont4:INT;
END_VAR
VAR PERSISTENT 
	PointerHistTablas:INT;
END_VAR

//                             >>>>>>>>>>>>>>>> Modelo de la tabla <<<<<<<<<<<<<<<<<

//Fin de producción 		
IF P_FinProduccion THEN 
Fin_Produccion();
END_IF;
IF P_EscribirModelo THEN
	ListFormatoTabla(); 
	Inicio_Nuevo_Modelo();
	
END_IF


//Envío de la linea de la tabla para el historico de control producción en el HMI del operario
 IF FlancFiltUpFtcEscHistTab.Q THEN 
	 EscStrHistoricoTablas();
 END_IF


Direccionamiento_variables_com();
FlancFiltUpFtcEscHistTab(CLK := FuncParoNodoCorteH4Remote1.Funci_CortHum4.tFiltro_up_Ftc.Q);

ACTION Direccionamiento_variables_com:
	//                           	>>>>>>>>>>>>>>>>>>>>>>>>>>>>      STRING      <<<<<<<<<<<<<<<<<<<<<<<<<<<<<<<<
    Var_Com_CH4_MulDis.aStringCom[80] := s_ModeloActualTabla;
	Var_Com_CH4_MulDis.aStringCom[81] := s_FormatoActualTabla;
	Var_Com_CH4_MulDis.aStringCom[82] := s_EspesorActualTabla;
	Var_Com_CH4_MulDis.aStringCom[83] := s_FechaInicModeloTab;
END_ACTION

METHOD EscStrHistoricoTablas : BOOL
VAR_INPUT
END_VAR
// Recorre todas las lineas de la tabla una posición y añade la nueva tabla en la linea 0 para mayor coodidad al visulizar

FOR PointerHistTablas := 100 TO 1 BY -1 DO 
	RegistroLocalDataBase.aHistoricStrTablasCH4[PointerHistTablas].ID := RegistroLocalDataBase.aHistoricStrTablasCH4[PointerHistTablas-1].ID;
	RegistroLocalDataBase.aHistoricStrTablasCH4[PointerHistTablas].Fecha := RegistroLocalDataBase.aHistoricStrTablasCH4[PointerHistTablas-1].Fecha;
	RegistroLocalDataBase.aHistoricStrTablasCH4[PointerHistTablas].Modelo := RegistroLocalDataBase.aHistoricStrTablasCH4[PointerHistTablas-1].Modelo;
	RegistroLocalDataBase.aHistoricStrTablasCH4[PointerHistTablas].Formato := RegistroLocalDataBase.aHistoricStrTablasCH4[PointerHistTablas-1].Formato;
	RegistroLocalDataBase.aHistoricStrTablasCH4[PointerHistTablas].Espesor :=RegistroLocalDataBase.aHistoricStrTablasCH4[PointerHistTablas-1].Espesor;
	RegistroLocalDataBase.aHistoricStrTablasCH4[PointerHistTablas].Maquina := RegistroLocalDataBase.aHistoricStrTablasCH4[PointerHistTablas-1].Maquina;
	RegistroLocalDataBase.aHistoricStrTablasCH4[PointerHistTablas].Cont_Piezas := RegistroLocalDataBase.aHistoricStrTablasCH4[PointerHistTablas-1].Cont_Piezas;
	RegistroLocalDataBase.aHistoricStrTablasCH4[PointerHistTablas].t_Entre_Piez_Ftc := RegistroLocalDataBase.aHistoricStrTablasCH4[PointerHistTablas-1].t_Entre_Piez_Ftc;
	RegistroLocalDataBase.aHistoricStrTablasCH4[PointerHistTablas].S_Justi_Paro_Ftc := RegistroLocalDataBase.aHistoricStrTablasCH4[PointerHistTablas-1].S_Justi_Paro_Ftc;
	
END_FOR
//Estructura de la array de la tabla para visualizar el historico de la tablas pasadas
RegistroLocalDataBase.aHistoricStrTablasCH4[0].ID := PointerHistTablas;
RegistroLocalDataBase.aHistoricStrTablasCH4[0].Fecha := Fecha_PLC.StringDateHourMin;
RegistroLocalDataBase.aHistoricStrTablasCH4[0].Modelo := FuncParoNodoCorteH4Remote1.sModeloActualTabla;
RegistroLocalDataBase.aHistoricStrTablasCH4[0].Formato := FuncParoNodoCorteH4Remote1.sFormatoActualTabla;
RegistroLocalDataBase.aHistoricStrTablasCH4[0].Espesor :=FuncParoNodoCorteH4Remote1.sEspesorActualTabla;
RegistroLocalDataBase.aHistoricStrTablasCH4[0].Maquina := 'Corte húmedo 4';
RegistroLocalDataBase.aHistoricStrTablasCH4[0].Cont_Piezas := FuncParoNodoCorteH4Remote1.Funci_CortHum4.Cont_Piezas_Ftc;
RegistroLocalDataBase.aHistoricStrTablasCH4[0].t_Entre_Piez_Ftc := FuncParoNodoCorteH4Remote1.Funci_CortHum4.t_Entre_Piez_Ftc;
RegistroLocalDataBase.aHistoricStrTablasCH4[0].S_Justi_Paro_Ftc := FuncParoNodoCorteH4Remote1.Funci_CortHum4.S_Justi_Paro_Ftc;
END_METHOD

METHOD Fin_Produccion : BOOL
VAR_INPUT	
END_VAR
var
	Puls_Fin_Produccion:BOOL;	
END_VAR
//Valores por defecto del modelo y fecha de inicio modelo

s_ModeloActualTabla:= 'Sin modelo de pieza';
s_ModeloEleccionTabla:= 'Sin modelo de pieza';
s_FormatoActualTabla:= 'Sin modelo de pieza';
s_FormatoEleccionTabla:= 'Sin modelo de pieza';
s_EspesorActualTabla:= 'Sin modelo de pieza';
s_EspesorEleccionTabla:= 'Sin modelo de pieza';
s_FechaInicModeloTab:= 'Sin modelo de pieza';
 
//Reset contador de piezas 
FuncParoNodoCorteH4Remote1.Funci_CortHum4.Fin_Produccion();
END_METHOD

METHOD Inicio_Nuevo_Modelo : BOOL
VAR_INPUT
END_VAR
VAR
END_VAR

// Envías la fecha de inicio modelo de tabla 
s_FechaInicModeloTab:=Fecha_PLC.Mes_Dia_Hora_Min_Real;

//Envías el modelo de la tabla de la variable preelección  
s_ModeloActualTabla:=s_ModeloEleccionTabla;
s_FormatoActualTabla:=s_FormatoEleccionTabla;
s_EspesorActualTabla:= s_EspesorEleccionTabla;
END_METHOD

METHOD ListFormatoTabla : BOOL
VAR_INPUT
END_VAR
// Función para poder realizar el desplegable de formato de la tabla en el Visu
IF IndexListFormatoTabla <> 6 THEN 
	IF IndexListFormatoTabla = 1 THEN 
		s_FormatoEleccionTabla:='17x17';
		Cont1:=Cont1+1;
	END_IF
	IF IndexListFormatoTabla = 2 THEN 
		s_FormatoEleccionTabla:='20x65';
		Cont2:=Cont2+1;
	END_IF
	IF IndexListFormatoTabla = 3 THEN 
		s_FormatoEleccionTabla:='30x15';
	END_IF
	IF IndexListFormatoTabla = 4 THEN 
		s_FormatoEleccionTabla:='30x30';
	END_IF
	IF IndexListFormatoTabla = 5 THEN 
		s_FormatoEleccionTabla:='03x03';
	END_IF

END_IF
END_METHOD

END_FUNCTION_BLOCK

// ---- POUs/PRGs_Nodos/FuncParoNodoMultidiscos.TcPOU
PROGRAM FuncParoNodoMultidiscos
VAR
	Funci_Multidiscos1:fb_Funciones_Paro;
	Funci_Multidiscos2:fb_Funciones_Paro;
	FunGeneMultidiscos1:FuncGeneralesMult1;
	FunGeneMultidiscos2:FuncGeneralesMult2;
	//Entradas Multidiscos1
	Ftc_Multidiscos1: BOOL;	
	ForzadoFtcMultidiscos1:BOOL;	
	Consenso_Multidiscos1: BOOL;
	//Entradas Multidiscos2
	Ftc2_Multidiscos2: BOOL;
	ForzadoFtc2_Multidiscos2: BOOL;
	Consenso_Multidiscos2: BOOL;
//Entradas Fotocelula libre 1
	Ftc3: BOOL;
	ForzadoFtc3: BOOL;
	Consenso3: BOOL;
//Entradas Fotocelula libre 2
	Ftc4: BOOL;
	ForzadoFtc4: BOOL;
	Consenso4: BOOL;
	
	Multidiscos1StrFuncParoEnviar:StrFuncParoEnviar;
	Multidiscos2StrFuncParoEnviar:StrFuncParoEnviar;
	Libre1StrFuncParoEnviar:StrFuncParoEnviar;
	Libre2StrFuncParoEnviar:StrFuncParoEnviar;	
END_VAR
VAR RETAIN
END_VAR
VAR_INPUT
//Multidiscos 1
	sFormatoEleccionTabla_MD1:STRING;
	sModeloEleccionTabla_MD1:STRING;
	sEspesorEleccionTabla_MD1:STRING;
//Multidiscos 2
	sFormatoEleccionTabla_MD2:STRING;
	sModeloEleccionTabla_MD2:STRING;
	sEspesorEleccionTabla_MD2:STRING;
END_VAR
VAR PERSISTENT 
	HMI_Tiempo_Offset_MParoMult1:INT:=3;
	HMI_Tiempo_Offset_MParoMult2:INT:=3;
	HMI_TiempoFiltradoFotMul_1:TIME:=T#1S;
	HMI_TiempoFiltradoFotMul_2:TIME:=T#1S;
// Generales multidoscos 1
	sModeloActualTabla_MD1:STRING;
	sFormatoActualTabla_MD1:STRING;
	sEspesorActualTabla_MD1:STRING;
	sFechaInicModeloTab_MD1:STRING;
// Generales multidoscos 2
	sModeloActualTabla_MD2:STRING;
	sFormatoActualTabla_MD2:STRING;
	sEspesorActualTabla_MD2:STRING;
	sFechaInicModeloTab_MD2:STRING;
END_VAR

//Funciones de paro para cada zona(Fotocelula)

//>>>>>>>>>>>>>>>>>>>>>>>>>>>>>>>>>>>>>>>>>>>>>         	Multidiscos 1         <<<<<<<<<<<<<<<<<<<<<<<<<<<<<<<<<<<<<<<<<<<<<<<<<<<<<<<<<<
Funci_Multidiscos1(Fotocelula:=Ftc_Multidiscos1 OR ForzadoFtcMultidiscos1, 
					Tiempo_Offset_MParo:=HMI_Tiempo_Offset_MParoMult1, 
					TiempoFiltradoFotocel:=HMI_TiempoFiltradoFotMul_1,
					_StrFuncParoEnviar => Multidiscos1StrFuncParoEnviar,);
					
//>>>>>>>>>>>>>>>>>>>>>>>>>>>>>>>>>>>>>>>>>>>>>         	Multidiscos 2        <<<<<<<<<<<<<<<<<<<<<<<<<<<<<<<<<<<<<<<<<<<<<<<<<<<<<<<<<<
Funci_Multidiscos2(Fotocelula:= Ftc2_Multidiscos2 OR ForzadoFtc2_Multidiscos2,
						Tiempo_Offset_MParo:=HMI_Tiempo_Offset_MParoMult2, 
						TiempoFiltradoFotocel:=HMI_TiempoFiltradoFotMul_2,
						_StrFuncParoEnviar => Multidiscos2StrFuncParoEnviar,);
						

										
Direccionamiento_variables_com();
Linkado_Entradas();
FunGeneMultidiscos1(s_ModeloActualTabla => sModeloActualTabla_MD1,s_ModeloEleccionTabla => sModeloEleccionTabla_MD1,s_FechaInicModeloTab=>sFechaInicModeloTab_MD1,s_FormatoActualTabla=>sFormatoActualTabla_MD1,s_FormatoEleccionTabla=>sFormatoEleccionTabla_MD1,s_EspesorActualTabla=>sEspesorActualTabla_MD1,s_EspesorEleccionTabla=>sEspesorEleccionTabla_MD1);
FunGeneMultidiscos2(s_ModeloActualTabla => sModeloActualTabla_MD2,s_ModeloEleccionTabla => sModeloEleccionTabla_MD2,s_FechaInicModeloTab=>sFechaInicModeloTab_MD2,s_FormatoActualTabla=>sFormatoActualTabla_MD2,s_FormatoEleccionTabla=>sFormatoEleccionTabla_MD2,s_EspesorActualTabla=>sEspesorActualTabla_MD2,s_EspesorEleccionTabla=>sEspesorEleccionTabla_MD2);

ACTION Direccionamiento_variables_com:
// Direccionamiento de las variables a la marca que les corresponde donde después se leeran desde el plc maestro



//								>>>>>>>>>>>>>>>>>>>>>>>>>>>>      WORDS    <<<<<<<<<<<<<<<<<<<<<<<<<<<<<<<<

	Var_Com_CH4_MulDis.aWordCom[0]:= INT_TO_WORD (Multidiscos1StrFuncParoEnviar.Cont_Piezas);	    //Contadores de cada fotocelula 
	Var_Com_CH4_MulDis.aWordCom[1]:= INT_TO_WORD (Multidiscos2StrFuncParoEnviar.Cont_Piezas);		//Contadores de cada fotocelula 
	Var_Com_CH4_MulDis.aWordCom[2]:= INT_TO_WORD (Libre1StrFuncParoEnviar.Cont_Piezas);		//Contadores de cada fotocelula 
	Var_Com_CH4_MulDis.aWordCom[3]:= INT_TO_WORD (Libre2StrFuncParoEnviar.Cont_Piezas);		//Contadores de cada fotocelula 
	Var_Com_CH4_MulDis.aWordCom[4]:= INT_TO_WORD (Multidiscos1StrFuncParoEnviar.Min_Parado_Ftc);			//Minutos actuales parado
	Var_Com_CH4_MulDis.aWordCom[5]:= INT_TO_WORD (Multidiscos2StrFuncParoEnviar.Min_Parado_Ftc);			//Minutos actuales parado
	Var_Com_CH4_MulDis.aWordCom[6]:= INT_TO_WORD (Libre1StrFuncParoEnviar.Min_Parado_Ftc);			//Minutos actuales parado
	Var_Com_CH4_MulDis.aWordCom[7]:= INT_TO_WORD (Libre2StrFuncParoEnviar.Min_Parado_Ftc);			//Minutos actuales parado
	
	
	
//                           	>>>>>>>>>>>>>>>>>>>>>>>>>>>>      TIME   <<<<<<<<<<<<<<<<<<<<<<<<<<<<<<<<
	
	
	Var_Com_CH4_MulDis.aTimeCom[0]:=  Multidiscos1StrFuncParoEnviar.t_Entre_Piez_Ftc; 			//Tiempo entre piezas
	Var_Com_CH4_MulDis.aTimeCom[1]:=  Multidiscos2StrFuncParoEnviar.t_Entre_Piez_Ftc;			//Tiempo entre piezas
	Var_Com_CH4_MulDis.aTimeCom[2]:= Libre1StrFuncParoEnviar.t_Entre_Piez_Ftc;				//Tiempo entre piezas
	Var_Com_CH4_MulDis.aTimeCom[3]:= Libre2StrFuncParoEnviar.t_Entre_Piez_Ftc;				//Tiempo entre piezas
	Var_Com_CH4_MulDis.aTimeCom[4]:= Multidiscos1StrFuncParoEnviar.t_Entr_Piez_Ante_Ftc; 		//Tiempo entre piezas anterior
	Var_Com_CH4_MulDis.aTimeCom[5]:= Multidiscos2StrFuncParoEnviar.t_Entr_Piez_Ante_Ftc; 		//Tiempo entre piezas anterior
	Var_Com_CH4_MulDis.aTimeCom[6]:= Libre1StrFuncParoEnviar.t_Entr_Piez_Ante_Ftc; 		//Tiempo entre piezas anterior
	Var_Com_CH4_MulDis.aTimeCom[7]:= Libre2StrFuncParoEnviar.t_Entr_Piez_Ante_Ftc; 		//Tiempo entre piezas anterior
	
	
	
	
//                           	>>>>>>>>>>>>>>>>>>>>>>>>>>>>      STRING  <<<<<<<<<<<<<<<<<<<<<<<<<<<<<<<<
    Var_Com_CH4_MulDis.aStringCom[0] := Multidiscos1StrFuncParoEnviar.H_InParo_Ftc;         //Hora inicio paro 
	Var_Com_CH4_MulDis.aStringCom[1] := Multidiscos2StrFuncParoEnviar.H_InParo_Ftc;         //Hora inicio paro 
	Var_Com_CH4_MulDis.aStringCom[2] := Libre1StrFuncParoEnviar.H_InParo_Ftc;         //Hora inicio paro 
	Var_Com_CH4_MulDis.aStringCom[3] := Libre2StrFuncParoEnviar.H_InParo_Ftc;         //Hora inicio paro 
	Var_Com_CH4_MulDis.aStringCom[4] := Multidiscos1StrFuncParoEnviar.H_FinParo_Ftc;        //Hora Fin paro 
	Var_Com_CH4_MulDis.aStringCom[5] := Multidiscos2StrFuncParoEnviar.H_FinParo_Ftc;        //Hora Fin paro 
	Var_Com_CH4_MulDis.aStringCom[6] := Libre1StrFuncParoEnviar.H_FinParo_Ftc;        //Hora Fin paro 
	Var_Com_CH4_MulDis.aStringCom[7] := Libre2StrFuncParoEnviar.H_FinParo_Ftc;        //Hora Fin paro 
	Var_Com_CH4_MulDis.aStringCom[8] := Multidiscos1StrFuncParoEnviar.S_Justi_Paro_Ftc;		//Justificación del paro
	Var_Com_CH4_MulDis.aStringCom[9] := Multidiscos2StrFuncParoEnviar.S_Justi_Paro_Ftc;		//Justificación del paro
	Var_Com_CH4_MulDis.aStringCom[10] := Libre1StrFuncParoEnviar.S_Justi_Paro_Ftc;		//Justificación del paro
	Var_Com_CH4_MulDis.aStringCom[11] := Libre2StrFuncParoEnviar.S_Justi_Paro_Ftc;		//Justificación del paro
	
	
//                           	>>>>>>>>>>>>>>>>>>>>>>>>>>>>      Bool  <<<<<<<<<<<<<<<<<<<<<<<<<<<<<<<<	

	Var_Com_CH4_MulDis.aBoolCom[0] := Multidiscos1StrFuncParoEnviar.Fotocelula;						//Fotocelula Real
	Var_Com_CH4_MulDis.aBoolCom[1] := Multidiscos2StrFuncParoEnviar.Fotocelula;						//Fotocelula Real
	Var_Com_CH4_MulDis.aBoolCom[2] := Libre1StrFuncParoEnviar.Fotocelula;						//Fotocelula Real
	Var_Com_CH4_MulDis.aBoolCom[3] := Libre2StrFuncParoEnviar.Fotocelula;						//Fotocelula Real
	Var_Com_CH4_MulDis.aBoolCom[4] := Multidiscos1StrFuncParoEnviar.MParo_Ftc;				//Marca de paro 
	Var_Com_CH4_MulDis.aBoolCom[5] := Multidiscos2StrFuncParoEnviar.MParo_Ftc;				//Marca de paro 
	Var_Com_CH4_MulDis.aBoolCom[6] := Libre1StrFuncParoEnviar.MParo_Ftc;				//Marca de paro 
	Var_Com_CH4_MulDis.aBoolCom[7] := Libre2StrFuncParoEnviar.MParo_Ftc;				//Marca de paro 
	Var_Com_CH4_MulDis.aBoolCom[8] := Multidiscos1StrFuncParoEnviar.M_SinParo_Ftc;			//Marca de sin paro activo
	Var_Com_CH4_MulDis.aBoolCom[9] := Multidiscos2StrFuncParoEnviar.M_SinParo_Ftc;			//Marca de sin paro activo
	Var_Com_CH4_MulDis.aBoolCom[10] := Libre1StrFuncParoEnviar.M_SinParo_Ftc;			//Marca de sin paro activo
	Var_Com_CH4_MulDis.aBoolCom[11] := Libre2StrFuncParoEnviar.M_SinParo_Ftc;			//Marca de sin paro activo
	Var_Com_CH4_MulDis.aBoolCom[12] := Multidiscos1StrFuncParoEnviar.tFiltro_up_Ftc;			//Q Temp Up Filtro Fotocelulas
	Var_Com_CH4_MulDis.aBoolCom[13] := Multidiscos2StrFuncParoEnviar.tFiltro_up_Ftc;			//Q Temp Up Filtro Fotocelulas
	Var_Com_CH4_MulDis.aBoolCom[14] := Libre1StrFuncParoEnviar.tFiltro_up_Ftc;			//Q Temp Up Filtro Fotocelulas
	Var_Com_CH4_MulDis.aBoolCom[15] := Libre2StrFuncParoEnviar.tFiltro_up_Ftc;			//Q Temp Up Filtro Fotocelulas
	Var_Com_CH4_MulDis.aBoolCom[16] := Multidiscos1StrFuncParoEnviar.tFiltro_down_Ftc;		//Q Temp Down Filtro Fotocelulas
	Var_Com_CH4_MulDis.aBoolCom[17] := Multidiscos2StrFuncParoEnviar.tFiltro_down_Ftc;		//Q Temp Down Filtro Fotocelulas
	Var_Com_CH4_MulDis.aBoolCom[18] := Libre1StrFuncParoEnviar.tFiltro_down_Ftc;		//Q Temp Down Filtro Fotocelulas
	Var_Com_CH4_MulDis.aBoolCom[19] := Libre2StrFuncParoEnviar.tFiltro_down_Ftc;		//Q Temp Down Filtro Fotocelulas
END_ACTION

ACTION Linkado_Entradas:
// Linkado entradas
Ftc_Multidiscos1:=     MAIN.id0Local.0;
Consenso_Multidiscos1:= TRUE;// main.id0Local2.1;


Ftc2_Multidiscos2:=      MAIN.id0Local.2;
Consenso_Multidiscos2:= TRUE;// main.id0Local2.3;


Ftc3:=      main.id0Local.4;
Consenso3:= TRUE;// main.id0Local2.5;


Ftc4:=      main.id0Local.6;
Consenso4:= TRUE;// main.id0Local2.7;
END_ACTION

END_PROGRAM

// ---- POUs/FBs/FuncGeneralesMult1.TcPOU
FUNCTION_BLOCK FuncGeneralesMult1
VAR_INPUT
IndexListFormatoTabla:INT;
END_VAR
VAR_OUTPUT
	//Modelo dividido en strings para DataBase
	s_ModeloActualTabla:STRING;
	s_FormatoActualTabla:STRING;
	s_EspesorActualTabla:STRING;
	s_ModeloEleccionTabla:STRING;
	s_FormatoEleccionTabla:STRING;
	s_EspesorEleccionTabla:STRING;
	//Comunes
	s_JustificaParoComun:STRING;
	s_FechaInicModeloTab:STRING;
END_VAR
VAR
	Reset_Fin_Prod:BOOL;
	P_FinProduccion:BOOL;
	P_EscribirModelo:BOOL;
	pul_Justif_Paro:BOOL;
	Cont1:INT;
	Cont2:INT;
	Cont3:INT;
	Cont4:INT;
END_VAR
VAR PERSISTENT 
END_VAR

//                             >>>>>>>>>>>>>>>> Modelo de la tabla <<<<<<<<<<<<<<<<<

//Fin de producción 		
IF P_FinProduccion THEN 
Fin_Produccion();
END_IF;
IF P_EscribirModelo THEN
	ListFormatoTabla(); 
	Inicio_Nuevo_Modelo();
	
END_IF


Direccionamiento_variables_com();

ACTION Direccionamiento_variables_com:
	//                           	>>>>>>>>>>>>>>>>>>>>>>>>>>>>      STRING      <<<<<<<<<<<<<<<<<<<<<<<<<<<<<<<<
    Var_Com_CH4_MulDis.aStringCom[84] := s_ModeloActualTabla;
	Var_Com_CH4_MulDis.aStringCom[85] := s_FormatoActualTabla;
	Var_Com_CH4_MulDis.aStringCom[86] := s_EspesorActualTabla;
	Var_Com_CH4_MulDis.aStringCom[87] := s_FechaInicModeloTab;
END_ACTION

METHOD Fin_Produccion : BOOL
VAR_INPUT	
END_VAR
var
	Puls_Fin_Produccion:BOOL;	
END_VAR
//Valores por defecto del modelo y fecha de inicio modelo

s_ModeloActualTabla:= 'Sin modelo de pieza';
s_ModeloEleccionTabla:= 'Sin modelo de pieza';
s_FormatoActualTabla:= 'Sin modelo de pieza';
s_FormatoEleccionTabla:= 'Sin modelo de pieza';
s_EspesorActualTabla:= 'Sin modelo de pieza';
s_EspesorEleccionTabla:= 'Sin modelo de pieza';
s_FechaInicModeloTab:= 'Sin modelo de pieza';
 
//Reset contador de piezas 
FuncParoNodoMultidiscos.Funci_Multidiscos1.Fin_Produccion();
END_METHOD

METHOD Inicio_Nuevo_Modelo : BOOL
VAR_INPUT
END_VAR
VAR
END_VAR

// Envías la fecha de inicio modelo de tabla 
s_FechaInicModeloTab:=Fecha_PLC.Mes_Dia_Hora_Min_Real;

//Envías el modelo de la tabla de la variable preelección  
s_ModeloActualTabla:=s_ModeloEleccionTabla;
s_FormatoActualTabla:=s_FormatoEleccionTabla;
s_EspesorActualTabla:= s_EspesorEleccionTabla;
END_METHOD

METHOD ListFormatoTabla : BOOL
VAR_INPUT
END_VAR
// Función para poder realizar el desplegable de formato de la tabla en el Visu
IF IndexListFormatoTabla <> 6 THEN 
	IF IndexListFormatoTabla = 1 THEN 
		s_FormatoEleccionTabla:='17x17';
		Cont1:=Cont1+1;
	END_IF
	IF IndexListFormatoTabla = 2 THEN 
		s_FormatoEleccionTabla:='20x65';
		Cont2:=Cont2+1;
	END_IF
	IF IndexListFormatoTabla = 3 THEN 
		s_FormatoEleccionTabla:='30x15';
	END_IF
	IF IndexListFormatoTabla = 4 THEN 
		s_FormatoEleccionTabla:='30x30';
	END_IF
	IF IndexListFormatoTabla = 5 THEN 
		s_FormatoEleccionTabla:='03x03';
	END_IF

END_IF
END_METHOD

END_FUNCTION_BLOCK

// ---- POUs/FBs/FuncGeneralesMult2.TcPOU
FUNCTION_BLOCK FuncGeneralesMult2
VAR_INPUT
IndexListFormatoTabla:INT;
END_VAR
VAR_OUTPUT
	//Modelo dividido en strings para DataBase
	s_ModeloActualTabla:STRING;
	s_FormatoActualTabla:STRING;
	s_EspesorActualTabla:STRING;
	s_ModeloEleccionTabla:STRING;
	s_FormatoEleccionTabla:STRING;
	s_EspesorEleccionTabla:STRING;
	//Comunes
	s_JustificaParoComun:STRING;
	s_FechaInicModeloTab:STRING;
END_VAR
VAR
	Reset_Fin_Prod:BOOL;
	P_FinProduccion:BOOL;
	P_EscribirModelo:BOOL;
	pul_Justif_Paro:BOOL;
	Cont1:INT;
	Cont2:INT;
	Cont3:INT;
	Cont4:INT;
END_VAR
VAR PERSISTENT 
END_VAR

//                             >>>>>>>>>>>>>>>> Modelo de la tabla <<<<<<<<<<<<<<<<<

//Fin de producción 		
IF P_FinProduccion THEN 
Fin_Produccion();
END_IF;
IF P_EscribirModelo THEN
	ListFormatoTabla(); 
	Inicio_Nuevo_Modelo();
	
END_IF


Direccionamiento_variables_com();

ACTION Direccionamiento_variables_com:
	//                           	>>>>>>>>>>>>>>>>>>>>>>>>>>>>      STRING      <<<<<<<<<<<<<<<<<<<<<<<<<<<<<<<<
    Var_Com_CH4_MulDis.aStringCom[88] := s_ModeloActualTabla;
	Var_Com_CH4_MulDis.aStringCom[89] := s_FormatoActualTabla;
	Var_Com_CH4_MulDis.aStringCom[90] := s_EspesorActualTabla;
	Var_Com_CH4_MulDis.aStringCom[91] := s_FechaInicModeloTab;
END_ACTION

METHOD Fin_Produccion : BOOL
VAR_INPUT	
END_VAR
var
	Puls_Fin_Produccion:BOOL;	
END_VAR
//Valores por defecto del modelo y fecha de inicio modelo

s_ModeloActualTabla:= 'Sin modelo de pieza';
s_ModeloEleccionTabla:= 'Sin modelo de pieza';
s_FormatoActualTabla:= 'Sin modelo de pieza';
s_FormatoEleccionTabla:= 'Sin modelo de pieza';
s_EspesorActualTabla:= 'Sin modelo de pieza';
s_EspesorEleccionTabla:= 'Sin modelo de pieza';
s_FechaInicModeloTab:= 'Sin modelo de pieza';
 
//Reset contador de piezas 
FuncParoNodoMultidiscos.Funci_Multidiscos2.Fin_Produccion();
END_METHOD

METHOD Inicio_Nuevo_Modelo : BOOL
VAR_INPUT
END_VAR
VAR
END_VAR

// Envías la fecha de inicio modelo de tabla 
s_FechaInicModeloTab:=Fecha_PLC.Mes_Dia_Hora_Min_Real;

//Envías el modelo de la tabla de la variable preelección  
s_ModeloActualTabla:=s_ModeloEleccionTabla;
s_FormatoActualTabla:=s_FormatoEleccionTabla;
s_EspesorActualTabla:= s_EspesorEleccionTabla;
END_METHOD

METHOD ListFormatoTabla : BOOL
VAR_INPUT
END_VAR
// Función para poder realizar el desplegable de formato de la tabla en el Visu
IF IndexListFormatoTabla <> 6 THEN 
	IF IndexListFormatoTabla = 1 THEN 
		s_FormatoEleccionTabla:='17x17';
		Cont1:=Cont1+1;
	END_IF
	IF IndexListFormatoTabla = 2 THEN 
		s_FormatoEleccionTabla:='20x65';
		Cont2:=Cont2+1;
	END_IF
	IF IndexListFormatoTabla = 3 THEN 
		s_FormatoEleccionTabla:='30x15';
	END_IF
	IF IndexListFormatoTabla = 4 THEN 
		s_FormatoEleccionTabla:='30x30';
	END_IF
	IF IndexListFormatoTabla = 5 THEN 
		s_FormatoEleccionTabla:='03x03';
	END_IF

END_IF
END_METHOD

END_FUNCTION_BLOCK

// ---- POUs/Events_Alarms/Events.TcPOU
PROGRAM Events
VAR
	fbEventosGenerales_PLC:Eventos_PLC;
	bResetArrayAvisos:BOOL;
	bClearEvents:BOOL;
END_VAR

//Eventos Linea 4

fbEventosGenerales_PLC(bClearEvents:=bClearEvents,bResetArrayAvisos:=bResetArrayAvisos);

END_PROGRAM

// ---- POUs/Events_Alarms/Eventos_PLC.TcPOU
FUNCTION_BLOCK Eventos_PLC 
VAR_INPUT
	bResetArrayAvisos:BOOL;
	bClearEvents:BOOL;
END_VAR
VAR_OUTPUT
END_VAR
VAR
	fbMessage : FB_TcMessage;
	fbAlarm : FB_TcAlarm;
	fbTcEventLogger: FB_TcEventLogger;
    ITcClearLoggedEventsSettings : I_TcClearLoggedEventsSettings;
	fbAdsReadEvents:FB_AdsReadEvents;
	ArrayAvisos:ARRAY [1..100] OF BOOL;
	ArrayAlarmas:ARRAY [1..100] OF BOOL;
	i:INT;
	FalloPrueba:BOOL;
	bReadEvent: BOOL;
	//Prueba
    bReadEvents          : BOOL;
    bClear               : BOOL;
END_VAR

//Llamadas de funciones 
Llamadas_Y_funciones();

//  >>>>>>>>>>>>>>>>>>>>>>>>>>>>>>>>>>>>> Avisos <<<<<<<<<<<<<<<<<<<<<<<<<<<<<<<<<<<<<<<<<<
//Los avisos solo son a modo informativo. 




//Aviso 1        Lectura a PLC a maestro deshabilitada
IF NOT MAIN_Orden_Lectura_PLCs.bHabilitaLectura_Maestro AND NOT ArrayAvisos[1] THEN 
	ArrayAvisos[1]:=TRUE;
	fbMessage.CreateEx(TC_Events.My_Events.Lectura_PLC_Maestro_deshabilitada, 0);
	SendAviso();
END_IF
//Aviso 2        Lectura a PLCs deshabilitada
IF NOT MAIN_Orden_Lectura_PLCs.bHabilitarLecturaDePLCs AND NOT ArrayAvisos[2] THEN 
	ArrayAvisos[2]:=TRUE;
	fbMessage.CreateEx(TC_Events.My_Events.LecturaPLCsDeshabilitada, 0);
	SendAviso();
END_IF


//  >>>>>>>>>>>>>>>>>>>>>>>>>>>>>>>>>>>>> Alarmas <<<<<<<<<<<<<<<<<<<<<<<<<<<<<<<<<<<<<<<<<<
//Son fallos críticos. 

//Alarma 1  Fallo comunicación con PLC Maestro
 IF Lectura_Maestro.fbLectura_a_PLC_Maestro.AlarmaFalloComunicacion  AND NOT ArrayAlarmas[1] THEN 
	ArrayAlarmas[1]:=TRUE;
	fbAlarm.CreateEx(TC_Events.My_Events.FalloLecturaPLC_Maestro, FALSE ,0);
	SendAlarma();
END_IF

//Alarma 2 Prueba 
IF FalloPrueba AND NOT ArrayAlarmas[2] THEN 
	ArrayAlarmas[2]:=TRUE;
	fbAlarm.CreateEx(TC_EVENTS.My_Events.Prueba,FALSE,0);
	SendAlarma();
END_IF

{warning 'add method implementation '}
METHOD BorraEventos : BOOL
fbTcEventLogger.ClearLoggedEvents(ipClearSettings:= ITcClearLoggedEventsSettings);
END_METHOD

ACTION Llamadas_Y_funciones:
//Reset array de los avisos    <<<<<<<<<<<<<<<   utilizados para que solo se envíe un mensaje y no esté continuamente enviando 
IF bResetArrayAvisos THEN 
	ResetArrayEvents();
END_IF

//Borrar avisos del HMI 
IF bClearEvents THEN 
	BorraEventos();
	ResetArrayEvents();
END_IF
END_ACTION

{warning 'add method implementation '}
METHOD ResetArrayEvents : BOOL
FOR i := 1 TO 100 BY 1 DO 
	ArrayAvisos[i]:= FALSE;
	ArrayAlarmas[i]:=FALSE;
END_FOR
END_METHOD

{warning 'add method implementation '}
METHOD SendAlarma : BOOL
fbAlarm.Raise(0);
END_METHOD

{warning 'add method implementation '}
METHOD SendAviso : BOOL
fbMessage.Send(0);
END_METHOD

END_FUNCTION_BLOCK

// ---- POUs/Funciones comunes/HMI.TcPOU
PROGRAM HMI
VAR

//OpenDialog:FbOpenDialog;
END_VAR

END_PROGRAM

// ---- GlobalTextList.TcGTLO
TEXTLIST GlobalTextList
  505 = '%i'
  650 = '%s'
  339 = '%S'
  429 = '%s \tContador fotocelula entrada horno inferior'
  862 = '%s \tContador fotocelula entrada horno superior'
  52 = '%s \tContador fotocelula entrada secadero'
  78 = '%s \tContador fotocelula salida airless 2'
  348 = '%s \tContador fotocelula salida prensa '
  177 = '%s \tContador piezas corte húmedo 4 '
  125 = '%s \tContador piezas multidiscos 1'
  699 = '%s \tContador piezas Multidiscos 1'
  246 = '%s \tContador piezas multidiscos 2'
  771 = '%s \tContador piezas Multidiscos 2'
  633 = '%t[s,ms]'
  577 = '//Quito las letras T# de la palabra a enviar\nt_Entre_Piez_Ftc := DELETE(t_Entre_Piez_Ftc, LEN := 2, POS := 1);'
  13 = 'Aceptar'
  1163 = 'ACEPTAR'
  1004 = 'Admin'
  801 = 'AJUSTES'
  152 = 'Ajustes'
  453 = 'Alarmas'
  259 = 'CAMBIO DE MODELO'
  856 = 'Contador de piezas'
  92 = 'Cont_Piezas'
  137 = 'Corte húmedo 4'
  1186 = 'CORTE HÚMEDO 4'
  448 = 'Delay Escritura'
  737 = 'Diagnostico'
  40 = 'Diagnostíco '
  35 = 'Diagnóstico'
  1366 = 'Día'
  29 = 'Elección modelo de la tabla CORTE HÚMEDO 4'
  16 = 'Elección modelo de la tabla LINEA 4'
  378 = 'Elección modelo de la tabla Multidiscos 1'
  634 = 'Elección modelo de la tabla Multidiscos 2'
  360 = 'Elige la opción de fin de producción \ndel modelo actual.'
  32 = 'En cuanto pulsas Reset paso a paso contadores se resetea \ncontador fotocelula salida prensa,\n  a los 10 min de no notar pieza en la entrada del secadero se resetea \ncontador entrada secadero,\n pasados 35 min sin notar pieza en salida airless 2 resetea \ncontador salida airless 2. \nA los 15 min que el contador de reset salida airless 2 se haya reseteado\n se resetea contador fotocelula entrada horno inferior. '
  172 = 'En cuanto se rearme la marcha se cerrará esta ventana.\nDe no haberte dado tiempo a justificar el paro deberas ir a \n"Registro tablas y justificación de paro" para introducirlo en la linea manualmente. '
  630 = 'En producción'
  432 = 'En producción todo OK'
  466 = 'Entre Piez %s'
  850 = 'Entre Piez Anterior %s'
  692 = 'Esmaltado'
  631 = 'Espesor'
  740 = 'ESPESOR'
  639 = 'Espesor de la tabla '
  765 = 'Exit'
  1002 = 'Fecha'
  394 = 'Fecha inicio del modelo actual'
  297 = 'Filtro Down'
  866 = 'Filtro Up'
  872 = 'Fin de producción'
  796 = 'Fin de producción del modelo'
  570 = 'Fin de producción temp'
  678 = 'Fin producción temporizado'
  550 = 'FINALIZAR'
  493 = 'Finalizar la producción\n mientras todavía quedan \npiezas por la línea \npero la prensa \nya ha parado.'
  806 = 'Finalizar la producción inmediatamente.\nNo deben haber tablas entre la prensa y\nel horno de destino.   '
  300 = 'Finalizar modelo'
  766 = 'FINALIZAR MODELO'
  419 = 'Formato'
  79 = 'FORMATO'
  215 = 'Formato de la tabla '
  884 = 'Forzar Fotocelula'
  998 = 'GreenCut'
  93 = 'Habilitar lectura a\nPLC CorteH4'
  841 = 'Habilitar lectura a\nPLC L4'
  332 = 'Habilitar lectura a\nPLCs'
  780 = 'Habilitar lectura al\nPLC'
  34 = 'Habilitar lectura al\nPLC Maestro'
  621 = 'Habilitar lectura del\nPLC Maestro'
  413 = 'Historial de las tablas CORTE HÚMEDO 4'
  532 = 'Histórico'
  907 = 'HISTÓRICO'
  248 = 'HISTÓRICO PRODUCCIÓN'
  681 = 'Hora Fin Paro'
  1204 = 'HORA INICIO'
  553 = 'Hora Inicio del paro'
  340 = 'Hora Inicio Paro'
  226 = 'Horno Inferior'
  412 = 'Horno Superior'
  1 = 'ID'
  867 = 'INICIADA:'
  179 = 'inicio'
  1088 = 'INICIO'
  1430 = 'INTRODUCE LOS DATOS DE LA OF'
  1183 = 'Justif paro'
  1000 = 'Justif paro '
  843 = 'Justific paro'
  1115 = 'Justifica brevemente el motivo del paro de la Linea.\nMáximo 5 palabras.'
  301 = 'Justificación del Paro'
  266 = 'JUSTIFICAR EL PARO ACTUAL'
  1158 = 'Justificar Paro'
  1063 = 'JUSTIFICAR PARO'
  366 = 'Línea  en paro'
  67 = 'Línea en paro'
  200 = 'Maquina'
  227 = 'Marca Paro '
  911 = 'Marca Sin Paro '
  316 = 'Min'
  209 = 'min'
  1127 = 'MINUTOS'
  914 = 'Minutos Parado'
  531 = 'Modelo'
  1198 = 'MODELO'
  735 = 'Modelo actual'
  12 = 'Modelo de la tabla '
  873 = 'MOTIVO 1'
  96 = 'Multidiscos'
  616 = 'Multidiscos '
  228 = 'Multidiscos 1'
  197 = 'MULTIDISCOS 1'
  118 = 'Multidiscos 2'
  989 = 'MULTIDISCOS 2'
  77 = 'Multidoscos'
  1014 = 'NINGÚN PARO ACTIVO'
  6 = 'None'
  1148 = 'NUEVO MODELO'
  1078 = 'Numero de Piezas'
  897 = 'Numero de tablas'
  1060 = 'Número de losas'
  364 = 'Número de piezas '
  700 = 'Número de tablas'
  86 = 'OF'
  1041 = 'Operario'
  23 = 'Operario_CH4'
  679 = 'Operario_Md1'
  1058 = 'Operario_Md2'
  1042 = 'ORDEN FABRICACIÓN -'
  490 = 'Paro activo'
  1136 = 'PARO ACTIVO'
  1107 = 'PARO ACTUAL'
  352 = 'PARO TOTAL'
  117 = 'PARO TOTAL '
  1678 = 'PARO TOTAL ACUMULADO '
  206 = 'PARO TOTAL DIARIO'
  566 = 'PAROS'
  21 = 'PARÁMETROS'
  1311 = 'PIEZAS'
  329 = 'Prensa'
  935 = 'PRODUCCIÓN'
  1123 = 'PRODUCCIÓN TURNO'
  258 = 'PRODUCIDAS'
  600 = 'Página de diagnóstico'
  732 = 'Reset contador'
  722 = 'Reset contador '
  20 = 'Reset paso a paso contadores'
  1413 = 'Revisa que no haya ninguna pieza en la línea.'
  224 = 'Ruta hacia horno'
  299 = 'Secadero'
  403 = 'Seg'
  59 = 'Selecciona la máquina con la que vas a trabajar'
  1182 = 'SELECCIONA LA SECCIÓN'
  225 = 'Sensor presencia tabla '
  864 = 'Si'
  1229 = 'Tablas'
  547 = 'TIEMPO DE PARO'
  510 = 'tiempo Entre Piez'
  64 = 'tiempo entre Piezas'
  906 = 'Tiempo entre Piezas'
  283 = 'Tiempo entre piezas'
  55 = 'Tiempo entre Piezas\nAnterior'
  571 = 'Tiempo entre tablas'
  966 = 'tiempo EntrePiez'
  705 = 'tiempo Entre_Piez'
  1056 = 'tiempo Entre_Piez_Ftc'
  649 = 'Tiempo filtrado fotocelulas\npara evitar parpadeos'
  501 = 'Tiempo para empezar \na contar como paro'
  433 = 'Total piezas'
  1284 = 'TOTAL PIEZAS'
  997 = 'Turno'
  173 = 'TURNO ACTUAL'
  371 = 'Vas a finalizar la producción de este modelo de tabla.\n¿Estas seguro que no queda ninguna tabla \nen la rodillera de entrada?'
  138 = 'Vas a finalizar la producción de este modelo de tabla.\n¿Estas seguro que no queda ninguna tabla \nen toda la línea?'
  58 = 'Vas a finalizar la producción de este modelo de tabla.\n¿Estas seguro que no queda ninguna tabla \nentre la prensa y la entrada del horno?'
  198 = 'Vas a finalizar la producción de este modelo.\n¿Estas seguro que no queda ninguna tabla \nen la rodillera de entrada?'
  1465 = 'Volver'
  1166 = 'VOLVER'
  729 = 'Zona entrada horno'
  278 = 'Zona presa'
  1577 = '¿Quieres finalizar el modelo?'
  506 = '¿Quieres finalizar la producción de este modelo?'
  1440 = '¿Quieres finalizar la producción?'
END_TEXTLIST

// ---- VISUs/Ajustes_Multidiscos1.TcVIS
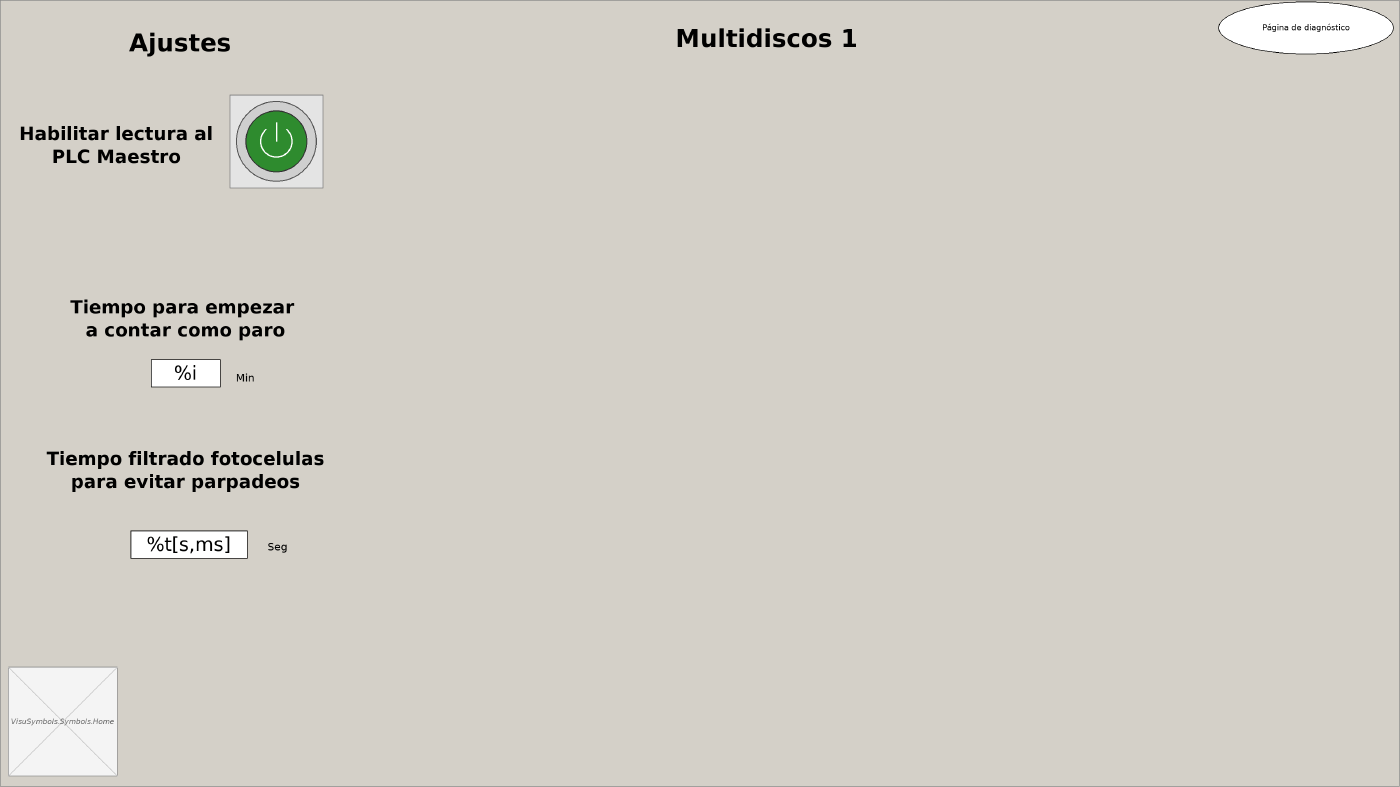
VISUALIZATION Ajustes_Multidiscos1  // 1920x1080
    Label (143,29 208x59), "Ajustes"
    Image (11,915 150x150), image: VisuSymbols.Symbols.Home
        OnMouseClick: change screen: Home_Multidis1
    Label (22,144 275x110), "Habilitar lectura al PLC Maestro"
    PowerSwitch (315,128 128x132), variable: MAIN_Orden_Lectura_PLCs.bHabilitaLectura_Maestro, behaviour: TOGGLE, style: Switch-PowerSwitch-Green
    Label (82,390 345x94), "Tiempo para empezar a contar como paro"
    Label (160,482 188x30)
    Rectangle (207,493 95x38), "%i", text variable: FuncParoNodoMultidiscos.HMI_Tiempo_Offset_MParoMult1
        OnMouseDown: write the text variable via Edit
    Label (307,500 59x37), "Min"
    Label (58,598 393x94), "Tiempo filtrado fotocelulas para evitar parpadeos"
    Label (351,732 59x37), "Seg"
    Rectangle (179,728 160x38), "%t[s,ms]", text variable: FuncParoNodoMultidiscos.HMI_TiempoFiltradoFotMul_1
        OnMouseDown: write the text variable via Edit
    Ellipse (1671,2 240x72), "Página de diagnóstico"
        OnMouseClick: change screen: DiagnosticoFB
    Label (884,23 335x59), "Multidiscos 1"
END_VISUALIZATION

// ---- VISUs/Ajustes_Multidiscos2.TcVIS
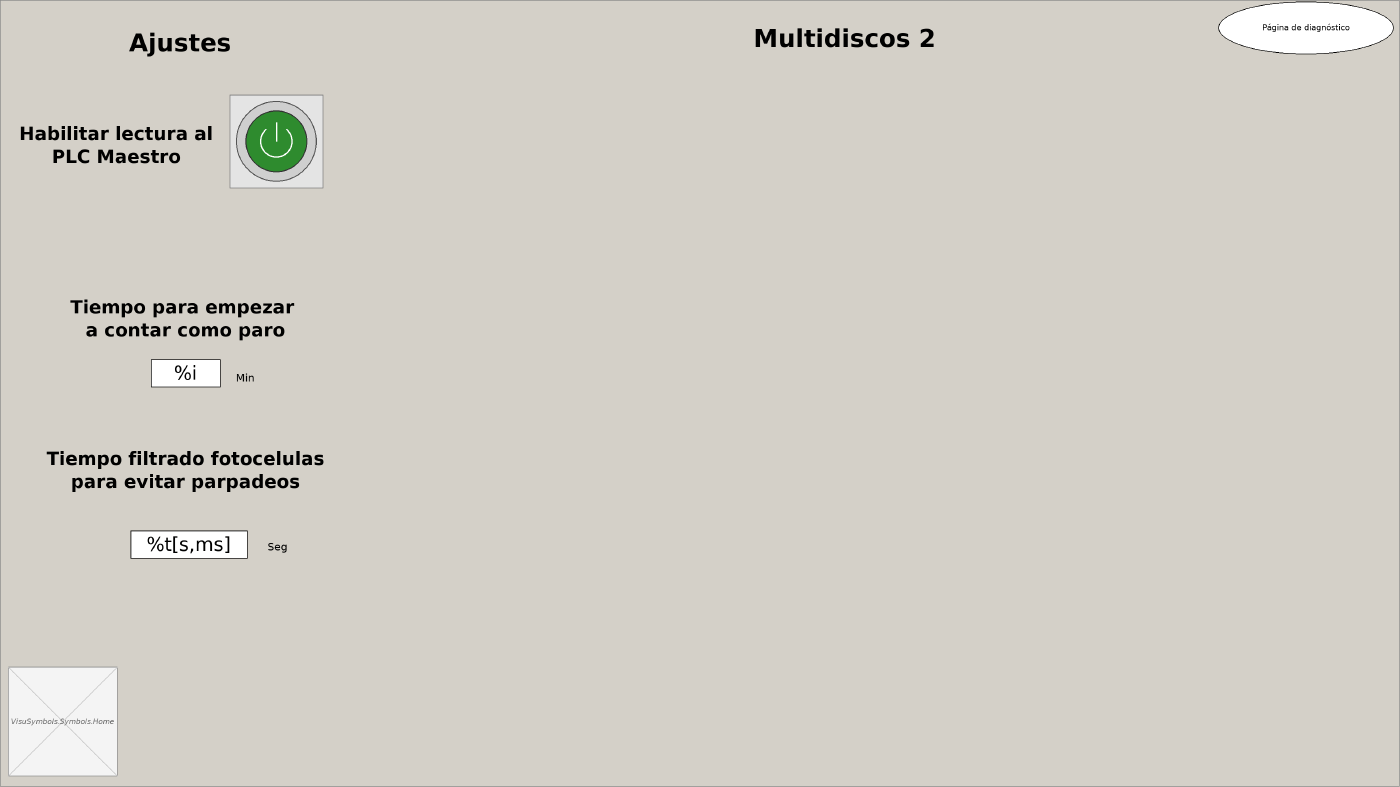
VISUALIZATION Ajustes_Multidiscos2  // 1920x1080
    Label (143,29 208x59), "Ajustes"
    Image (11,915 150x150), image: VisuSymbols.Symbols.Home
        OnMouseClick: change screen: Home_Multidis2
    Label (22,144 275x110), "Habilitar lectura al PLC Maestro"
    PowerSwitch (315,128 128x132), variable: MAIN_Orden_Lectura_PLCs.bHabilitaLectura_Maestro, behaviour: TOGGLE, style: Switch-PowerSwitch-Green
    Label (82,390 345x94), "Tiempo para empezar a contar como paro"
    Label (160,482 188x30)
    Rectangle (207,493 95x38), "%i", text variable: FuncParoNodoMultidiscos.HMI_Tiempo_Offset_MParoMult2
        OnMouseDown: write the text variable via Edit
    Label (307,500 59x37), "Min"
    Label (58,598 393x94), "Tiempo filtrado fotocelulas para evitar parpadeos"
    Label (351,732 59x37), "Seg"
    Rectangle (179,728 160x38), "%t[s,ms]", text variable: FuncParoNodoMultidiscos.HMI_TiempoFiltradoFotMul_2
        OnMouseDown: write the text variable via Edit
    Label (991,23 335x59), "Multidiscos 2"
    Ellipse (1671,2 240x72), "Página de diagnóstico"
        OnMouseClick: change screen: DiagnosticoFB
END_VISUALIZATION

// ---- VISUs/DiagnosticoFB.TcVIS
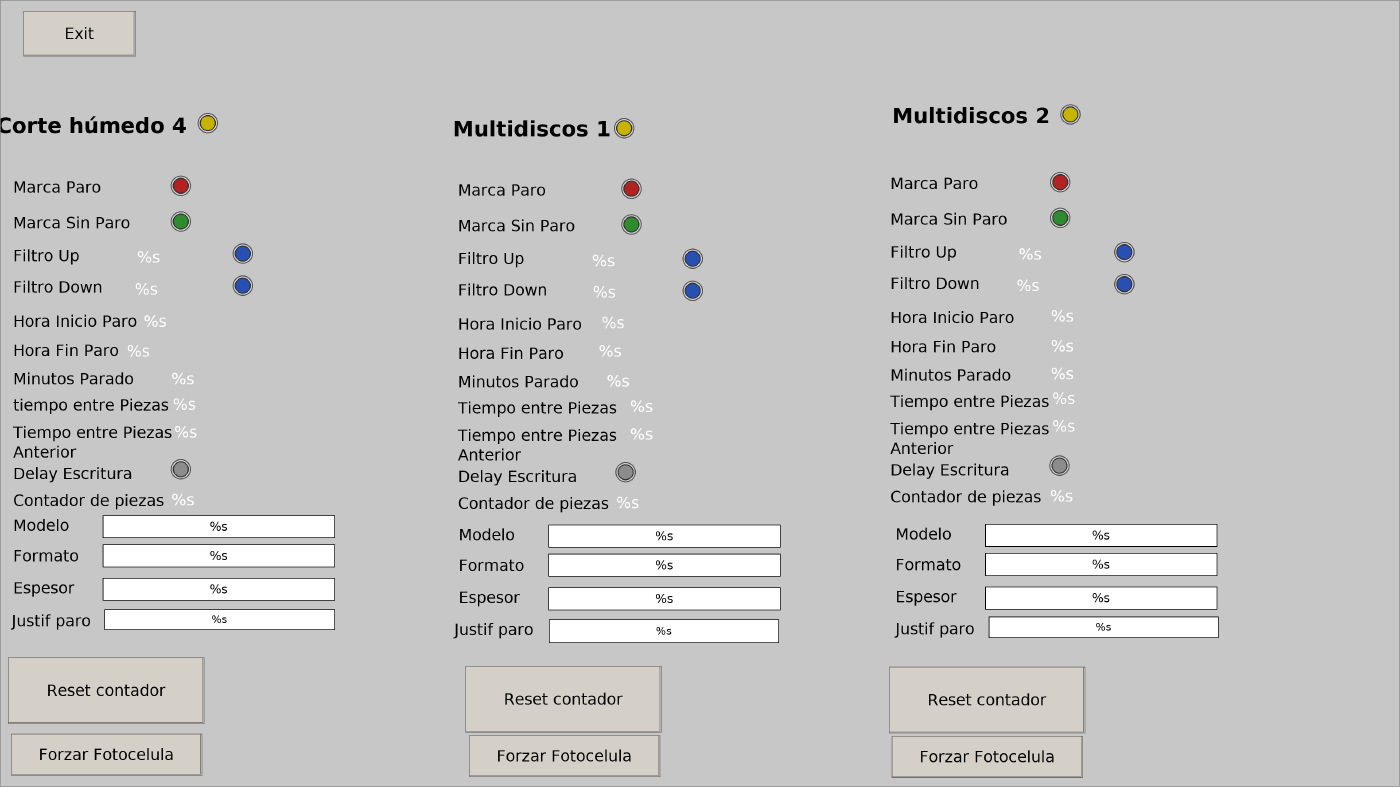
VISUALIZATION DiagnosticoFB  // 1920x1080
    Rectangle (185,338 93x30), "%s", text variable: FuncParoNodoCorteH4Remote1.Funci_CortHum4.tFiltro_up_Ftc.ET
    Label (10,146 231x53), "Corte húmedo 4"
    Label (15,242 150x30), "Marca Paro"
    Lamp1 (269,153 32x32), variable: FuncParoNodoCorteH4Remote1.Funci_CortHum4.Fotocelula, style: Lamp-Lamp1-Yellow
    Lamp1 (232,239 32x32), variable: FuncParoNodoCorteH4Remote1.Funci_CortHum4.MParo_Ftc, style: Lamp-Lamp1-Red
    Label (15,291 188x30), "Marca Sin Paro"
    Lamp1 (232,288 32x32), variable: FuncParoNodoCorteH4Remote1.Funci_CortHum4.M_SinParo_Ftc, style: Lamp-Lamp1-Green
    Label (15,336 117x30), "Filtro Up"
    Rectangle (182,382 93x30), "%s", text variable: FuncParoNodoCorteH4Remote1.Funci_CortHum4.tFiltro_down_Ftc.ET
    Label (15,379 143x30), "Filtro Down"
    Rectangle (194,426 183x30), "%s", text variable: FuncParoNodoCorteH4Remote1.Funci_CortHum4.H_InParo_Ftc
    Label (15,426 204x30), "Hora Inicio Paro"
    Lamp1 (317,332 32x32), variable: FuncParoNodoCorteH4Remote1.Funci_CortHum4.tFiltro_up_Ftc.Q, style: Lamp-Lamp1-Blue
    Lamp1 (317,376 32x32), variable: FuncParoNodoCorteH4Remote1.Funci_CortHum4.tFiltro_down_Ftc.Q, style: Lamp-Lamp1-Blue
    Rectangle (171,467 179x30), "%s", text variable: FuncParoNodoCorteH4Remote1.Funci_CortHum4.H_FinParo_Ftc
    Label (15,466 204x30), "Hora Fin Paro"
    Rectangle (232,505 192x30), "%s", text variable: FuncParoNodoCorteH4Remote1.Funci_CortHum4.Min_Parado_Ftc
    Label (15,505 204x30), "Minutos Parado"
    Label (15,541 244x30), "tiempo entre Piezas"
    Label (15,576 255x62), "Tiempo entre Piezas Anterior"
    Label (15,635 204x30), "Delay Escritura"
    Rectangle (232,671 93x30), "%s", text variable: FuncParoNodoCorteH4Remote1.Funci_CortHum4.Cont_Piezas_Ftc
    Label (15,672 215x30), "Contador de piezas"
    Lamp1 (232,628 32x32), variable: FuncParoNodoCorteH4Remote1.Funci_CortHum4.Delay_Esc_Ftc.Q, style: Lamp-Lamp1-Gray
    Button (32,15 154x62), "Exit"
        OnMouseClick: change screen: Home_CortH4
    Rectangle (809,343 93x30), "%s", text variable: FuncParoNodoMultidiscos.Funci_Multidiscos1.tFiltro_up_Ftc.ET
    Label (614,134 231x86), "Multidiscos 1"
    Label (625,246 150x30), "Marca Paro"
    Lamp1 (840,160 32x32), variable: FuncParoNodoMultidiscos.Funci_Multidiscos1.Fotocelula, style: Lamp-Lamp1-Yellow
    Lamp1 (850,243 32x32), variable: FuncParoNodoMultidiscos.Funci_Multidiscos1.MParo_Ftc, style: Lamp-Lamp1-Red
    Label (625,295 188x30), "Marca Sin Paro"
    Lamp1 (850,292 32x32), variable: FuncParoNodoMultidiscos.Funci_Multidiscos1.M_SinParo_Ftc, style: Lamp-Lamp1-Green
    Label (625,340 117x30), "Filtro Up"
    Rectangle (810,386 93x30), "%s", text variable: FuncParoNodoMultidiscos.Funci_Multidiscos1.tFiltro_down_Ftc.ET
    Label (625,383 143x30), "Filtro Down"
    Rectangle (822,428 183x30), "%s", text variable: FuncParoNodoMultidiscos.Funci_Multidiscos1.H_InParo_Ftc
    Label (625,430 204x30), "Hora Inicio Paro"
    Lamp1 (934,339 32x32), variable: FuncParoNodoMultidiscos.Funci_Multidiscos1.tFiltro_up_Ftc.Q, style: Lamp-Lamp1-Blue
    Lamp1 (934,383 32x32), variable: FuncParoNodoMultidiscos.Funci_Multidiscos1.tFiltro_down_Ftc.Q, style: Lamp-Lamp1-Blue
    Rectangle (818,467 179x30), "%s", text variable: FuncParoNodoMultidiscos.Funci_Multidiscos1.H_FinParo_Ftc
    Label (625,470 204x30), "Hora Fin Paro"
    Rectangle (829,508 192x30), "%s", text variable: FuncParoNodoMultidiscos.Funci_Multidiscos1.Min_Parado_Ftc
    Label (625,509 204x30), "Minutos Parado"
    Label (625,545 244x30), "Tiempo entre Piezas"
    Label (625,580 255x62), "Tiempo entre Piezas Anterior"
    Label (625,639 204x30), "Delay Escritura"
    Rectangle (842,675 93x30), "%s", text variable: FuncParoNodoMultidiscos.Funci_Multidiscos1.Cont_Piezas_Ftc
    Label (625,676 215x30), "Contador de piezas"
    Lamp1 (842,632 32x32), variable: FuncParoNodoMultidiscos.Funci_Multidiscos1.Delay_Esc_Ftc.Q, style: Lamp-Lamp1-Gray
    Rectangle (1394,334 93x30), "%s", text variable: FuncParoNodoMultidiscos.Funci_Multidiscos2.tFiltro_up_Ftc.ET
    Label (1207,115 250x88), "Multidiscos 2"
    Label (1218,237 150x30), "Marca Paro"
    Lamp1 (1452,141 32x32), variable: FuncParoNodoMultidiscos.Funci_Multidiscos2.Fotocelula, style: Lamp-Lamp1-Yellow
    Lamp1 (1438,234 32x32), variable: FuncParoNodoMultidiscos.Funci_Multidiscos2.MParo_Ftc, style: Lamp-Lamp1-Red
    Label (1218,286 188x30), "Marca Sin Paro"
    Lamp1 (1438,283 32x32), variable: FuncParoNodoMultidiscos.Funci_Multidiscos2.M_SinParo_Ftc, style: Lamp-Lamp1-Green
    Label (1218,331 117x30), "Filtro Up"
    Rectangle (1391,377 93x30), "%s", text variable: FuncParoNodoMultidiscos.Funci_Multidiscos2.tFiltro_down_Ftc.ET
    Label (1218,374 143x30), "Filtro Down"
    Rectangle (1438,419 183x30), "%s", text variable: FuncParoNodoMultidiscos.Funci_Multidiscos2.H_InParo_Ftc
    Label (1218,421 204x30), "Hora Inicio Paro"
    Lamp1 (1526,330 32x32), variable: FuncParoNodoMultidiscos.Funci_Multidiscos2.tFiltro_up_Ftc.Q, style: Lamp-Lamp1-Blue
    Lamp1 (1526,374 32x32), variable: FuncParoNodoMultidiscos.Funci_Multidiscos2.tFiltro_down_Ftc.Q, style: Lamp-Lamp1-Blue
    Rectangle (1438,460 179x30), "%s", text variable: FuncParoNodoMultidiscos.Funci_Multidiscos2.H_FinParo_Ftc
    Label (1218,461 204x30), "Hora Fin Paro"
    Rectangle (1438,498 192x30), "%s", text variable: FuncParoNodoMultidiscos.Funci_Multidiscos2.Min_Parado_Ftc
    Label (1218,500 204x30), "Minutos Parado"
    Label (1218,536 244x30), "Tiempo entre Piezas"
    Label (1218,571 255x62), "Tiempo entre Piezas Anterior"
    Label (1218,630 204x30), "Delay Escritura"
    Rectangle (1437,666 93x30), "%s", text variable: FuncParoNodoMultidiscos.Funci_Multidiscos2.Cont_Piezas_Ftc
    Label (1218,667 215x30), "Contador de piezas"
    Lamp1 (1437,623 32x32), variable: FuncParoNodoMultidiscos.Funci_Multidiscos2.Delay_Esc_Ftc.Q, style: Lamp-Lamp1-Gray
    Rectangle (234,540 192x30), "%s", text variable: FuncParoNodoCorteH4Remote1.Funci_CortHum4.t_Entre_Piez_Ftc
    Rectangle (861,543 192x30), "%s", text variable: FuncParoNodoMultidiscos.Funci_Multidiscos1.t_Entre_Piez_Ftc
    Rectangle (1440,532 192x30), "%s", text variable: FuncParoNodoMultidiscos.Funci_Multidiscos2.t_Entre_Piez_Ftc
    Rectangle (236,578 192x30), "%s", text variable: FuncParoNodoCorteH4Remote1.Funci_CortHum4.t_Entr_Piez_Ante_Ftc
    Rectangle (861,581 192x30), "%s", text variable: FuncParoNodoMultidiscos.Funci_Multidiscos1.t_Entr_Piez_Ante_Ftc
    Rectangle (1440,570 192x30), "%s", text variable: FuncParoNodoMultidiscos.Funci_Multidiscos2.t_Entr_Piez_Ante_Ftc
    Button (11,902 269x91), "Reset contador"
        tap FuncParoNodoCorteH4Remote1.Funci_CortHum4.ResetContPiez
    Button (638,914 269x91), "Reset contador"
        tap FuncParoNodoMultidiscos.Funci_Multidiscos1.ResetContPiez
    Button (1219,915 269x91), "Reset contador"
        tap FuncParoNodoMultidiscos.Funci_Multidiscos2.ResetContPiez
    Button (643,1009 262x57), "Forzar Fotocelula"
        tap FuncParoNodoMultidiscos.ForzadoFtcMultidiscos1
    Button (1223,1010 262x57), "Forzar Fotocelula"
        tap FuncParoNodoMultidiscos.ForzadoFtc2_Multidiscos2
    Button (15,1007 262x57), "Forzar Fotocelula"
        tap FuncParoNodoCorteH4Remote1.ForzadoFtcCortHum4
    Label (15,706 92x30), "Modelo"
    Label (15,748 105x30), "Formato"
    Label (15,792 99x30), "Espesor"
    Rectangle (141,707 318x31), "%s", text variable: FuncParoNodoCorteH4Remote1.FunGeneCortHum4.s_ModeloActualTabla
        OnMouseDown: write the text variable via Edit
    Rectangle (141,747 318x31), "%s", text variable: FuncParoNodoCorteH4Remote1.FunGeneCortHum4.s_FormatoActualTabla
        OnMouseDown: write the text variable via Edit
    Rectangle (141,793 318x31), "%s", text variable: FuncParoNodoCorteH4Remote1.FunGeneCortHum4.s_EspesorActualTabla
        OnMouseDown: write the text variable via Edit
    Label (626,719 92x30), "Modelo"
    Label (626,761 105x30), "Formato"
    Label (626,805 99x30), "Espesor"
    Rectangle (752,720 318x31), "%s", text variable: FuncParoNodoMultidiscos.FunGeneMultidiscos1.s_ModeloActualTabla
        OnMouseDown: write the text variable via Edit
    Rectangle (752,760 318x31), "%s", text variable: FuncParoNodoMultidiscos.FunGeneMultidiscos1.s_FormatoActualTabla
        OnMouseDown: write the text variable via Edit
    Rectangle (752,806 318x31), "%s", text variable: FuncParoNodoMultidiscos.FunGeneMultidiscos1.s_EspesorActualTabla
        OnMouseDown: write the text variable via Edit
    Label (1225,718 92x30), "Modelo"
    Label (1225,760 105x30), "Formato"
    Label (1225,804 99x30), "Espesor"
    Rectangle (1351,719 318x31), "%s", text variable: FuncParoNodoMultidiscos.FunGeneMultidiscos2.s_ModeloActualTabla
        OnMouseDown: write the text variable via Edit
    Rectangle (1351,759 318x31), "%s", text variable: FuncParoNodoMultidiscos.FunGeneMultidiscos2.s_FormatoActualTabla
        OnMouseDown: write the text variable via Edit
    Rectangle (1351,805 318x31), "%s", text variable: FuncParoNodoMultidiscos.FunGeneMultidiscos2.s_EspesorActualTabla
        OnMouseDown: write the text variable via Edit
    Label (13,837 123x30), "Justif paro"
    Rectangle (143,836 316x28), "%s", text variable: FuncParoNodoCorteH4Remote1.Funci_CortHum4.S_Justi_Paro_Ftc
        OnMouseDown: write the text variable via Edit
    Rectangle (753,850 315x32), "%s", text variable: FuncParoNodoMultidiscos.Funci_Multidiscos1.S_Justi_Paro_Ftc
        OnMouseDown: write the text variable via Edit
    Label (620,849 123x30), "Justif paro"
    Label (1225,848 123x30), "Justif paro"
    Rectangle (1356,846 315x29), "%s", text variable: FuncParoNodoMultidiscos.Funci_Multidiscos2.S_Justi_Paro_Ftc
        OnMouseDown: write the text variable via Edit
END_VISUALIZATION

// ---- VISUs/Home_CortH4.TcVIS
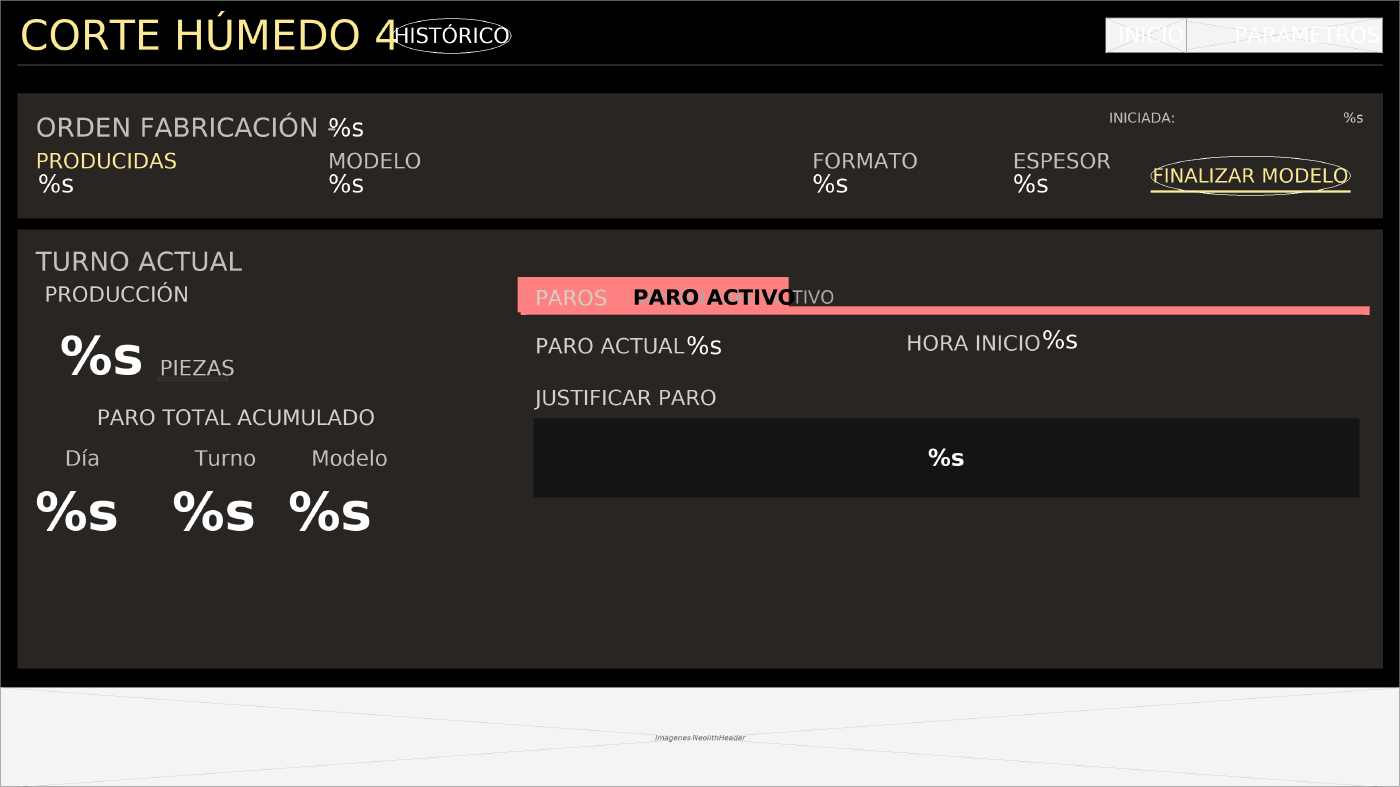
VISUALIZATION Home_CortH4  // 1920x1080
    Rectangle (24,315 1872x602)
    Rectangle (24,128 1872x171)
    Rectangle (24,88 1872x2)
    Ellipse (2013,684 456x77), "Fin de producción del modelo"
        OnMouseClick: OpenDialog Dialog=V_Emerg_Fin_Prod_Ch4, OpenModal=True, OpenCentered=True
    Label (24,16 514x64), "CORTE HÚMEDO 4"
    Lamp1 (2002,406 94x97), variable: FuncParoNodoCorteH4Remote1.Funci_CortHum4.Fotocelula, style: Lamp-Lamp1-Yellow
    Rectangle (1426,451 183x30), "%s", text variable: FuncParoNodoCorteH4Remote1.Funci_CortHum4.H_InParo_Ftc, invisible if: FuncParoNodoCorteH4Remote1.Funci_CortHum4.M_SinParo_Ftc
    Rectangle (938,459 192x30), "%s", text variable: FuncParoNodoCorteH4Remote1.Funci_CortHum4.Min_Parado_Ftc, invisible if: FuncParoNodoCorteH4Remote1.Funci_CortHum4.M_SinParo_Ftc
    Label (1949,260 244x30), "Tiempo entre Piezas"
    Label (1938,296 255x62), "Tiempo entre Piezas Anterior"
    Rectangle (2190,260 192x30), "%s", text variable: FuncParoNodoCorteH4Remote1.Funci_CortHum4.t_Entre_Piez_Ftc
    Rectangle (2190,312 192x30), "%s", text variable: FuncParoNodoCorteH4Remote1.Funci_CortHum4.t_Entr_Piez_Ante_Ftc
    Label (46,148 390x54), "ORDEN FABRICACIÓN -"
    Rectangle (1573,147 300x30), "%s", text variable: FuncParoNodoCorteH4Remote1.sFechaInicModeloTab
    Label (1518,147 99x30), "INICIADA:"
    Rectangle (732,574 1132x108), "%s", text variable: FuncParoNodoCorteH4Remote1.Funci_CortHum4.S_Justi_Paro_Ftc, invisible if: FuncParoNodoCorteH4Remote1.Funci_CortHum4.M_SinParo_Ftc
        OnMouseDown: write the text variable via Edit
    Image (116,-391 250x250), invisible if: FuncParoNodoCorteH4Remote1.Funci_CortHum4.M_SinParo_Ftc, image: ImagePool.Exclamación
    Image (454,-421 250x250), invisible if: FuncParoNodoCorteH4Remote1.Funci_CortHum4.M_SinParo_Ftc, image: ImagePool.Exclamación
    Image (1128,-383 250x250), invisible if: FuncParoNodoCorteH4Remote1.Funci_CortHum4.M_SinParo_Ftc, image: ImagePool.Exclamación
    Image (123,-961 250x250), invisible if: FuncParoNodoCorteH4Remote1.Funci_CortHum4.M_SinParo_Ftc, image: ImagePool.Exclamación
    Image (1136,-683 250x250), invisible if: FuncParoNodoCorteH4Remote1.Funci_CortHum4.M_SinParo_Ftc, image: ImagePool.Exclamación
    Image (478,-696 250x250), invisible if: FuncParoNodoCorteH4Remote1.Funci_CortHum4.M_SinParo_Ftc, image: ImagePool.Exclamación
    Image (1691,-991 250x250), invisible if: FuncParoNodoCorteH4Remote1.Funci_CortHum4.M_SinParo_Ftc, image: ImagePool.Exclamación
    Image (1600,24 296x48), "PARÁMETROS"
        OnMouseClick: change screen: Ajustes_CorteH4
    Image (1516,24 111x48), "INICIO"
        OnMouseClick: change screen: Home_Sel_Maq
    Ellipse (2006,785 456x77), "Histórico"
        OnMouseClick: change screen: HistTablaTablas_Ch4
    Group (447,203 1095x69)
        Rectangle (0,29 671x40), "%s", text variable: FuncParoNodoCorteH4Remote1.sModeloActualTabla
        Rectangle (939,29 120x40), "%s", text variable: FuncParoNodoCorteH4Remote1.sEspesorActualTabla
        Rectangle (664,29 321x40), "%s", text variable: FuncParoNodoCorteH4Remote1.sFormatoActualTabla
        Label (0,0 487x36), "MODELO"
        Label (664,0 156x36), "FORMATO"
        Label (939,0 156x36), "ESPESOR"
    Rectangle (447,155 321x40), "%s", text variable: FuncParoNodoCorteH4Remote1.sFormatoActualTabla
    Label (46,203 199x36), "PRODUCIDAS"
    Rectangle (49,232 248x40), "%s", text variable: FuncParoNodoCorteH4Remote1.CortHum4StrFuncParoEnviar.Cont_Piezas
    Group (1578,214 274x54)
        Rectangle (0,47 274x3)
        Ellipse (0,0 274x54), "FINALIZAR MODELO"
            OnMouseClick: OpenDialog Dialog=V_Emerg_Fin_Prod_Ch4, OpenModal=True, OpenCentered=True
    Label (46,332 390x54), "TURNO ACTUAL"
    Label (58,386 199x36), "PRODUCCIÓN"
    Label (731,457 261x36), "PARO ACTUAL"
    Label (1240,453 261x36), "HORA INICIO"
    Group (1957,542 1116x80)
        RoundedRectangle (0,0 264x80), "MOTIVO 1"
        RoundedRectangle (284,0 264x80), "MOTIVO 1"
        RoundedRectangle (568,0 264x80), "MOTIVO 1"
        RoundedRectangle (852,0 264x80), "MOTIVO 1"
    Group (79,444 243x88)
        Rectangle (0,0 183x88), "%s", text variable: FuncParoNodoCorteH4Remote1.Funci_CortHum4.Cont_Piezas_Ftc
        Label (137,43 106x36), "PIEZAS"
        Rectangle (137,74 96x4), colour toggle: FuncParoNodoCorteH4Remote1.Funci_CortHum4.Fotocelula
    Label (731,528 261x36), "JUSTIFICAR PARO"
    Group (710,380 1168x48)
        Rectangle (4,44 1164x4)
        Rectangle (0,0 371x48)
        Label (21,11 199x36), "PAROS"
        Label (155,13 326x30), "NINGÚN PARO ACTIVO", invisible if: FuncParoNodoCorteH4Remote1.Funci_CortHum4.MParo_Ftc
        Label (155,13 235x30), "PARO ACTIVO", invisible if: FuncParoNodoCorteH4Remote1.Funci_CortHum4.M_SinParo_Ftc
    Ellipse (538,25 163x48), "HISTÓRICO"
        OnMouseClick: change screen: HistTablaTablas_Ch4
    Label (130,555 367x36), "PARO TOTAL ACUMULADO"
    Rectangle (45,658 183x88), "%s", text variable: FuncParoNodoCorteH4Remote1.Funci_CortHum4.t_Paro_Acumulado_Diario
    Label (86,611 76x36), "Día"
    Image (-3,943 1927x139), image: Imagenes.NeolithHeader
    Rectangle (233,658 167x88), "%s", text variable: FuncParoNodoCorteH4Remote1.Funci_CortHum4.t_Paro_Acumulado_Turno
    Label (264,611 102x36), "Turno"
    Rectangle (392,658 183x88), "%s", text variable: FuncParoNodoCorteH4Remote1.Funci_CortHum4.t_Paro_Acumulado_Modelo
    Label (424,611 118x36), "Modelo"
END_VISUALIZATION

// ---- VISUs/Home_Multidis1.TcVIS
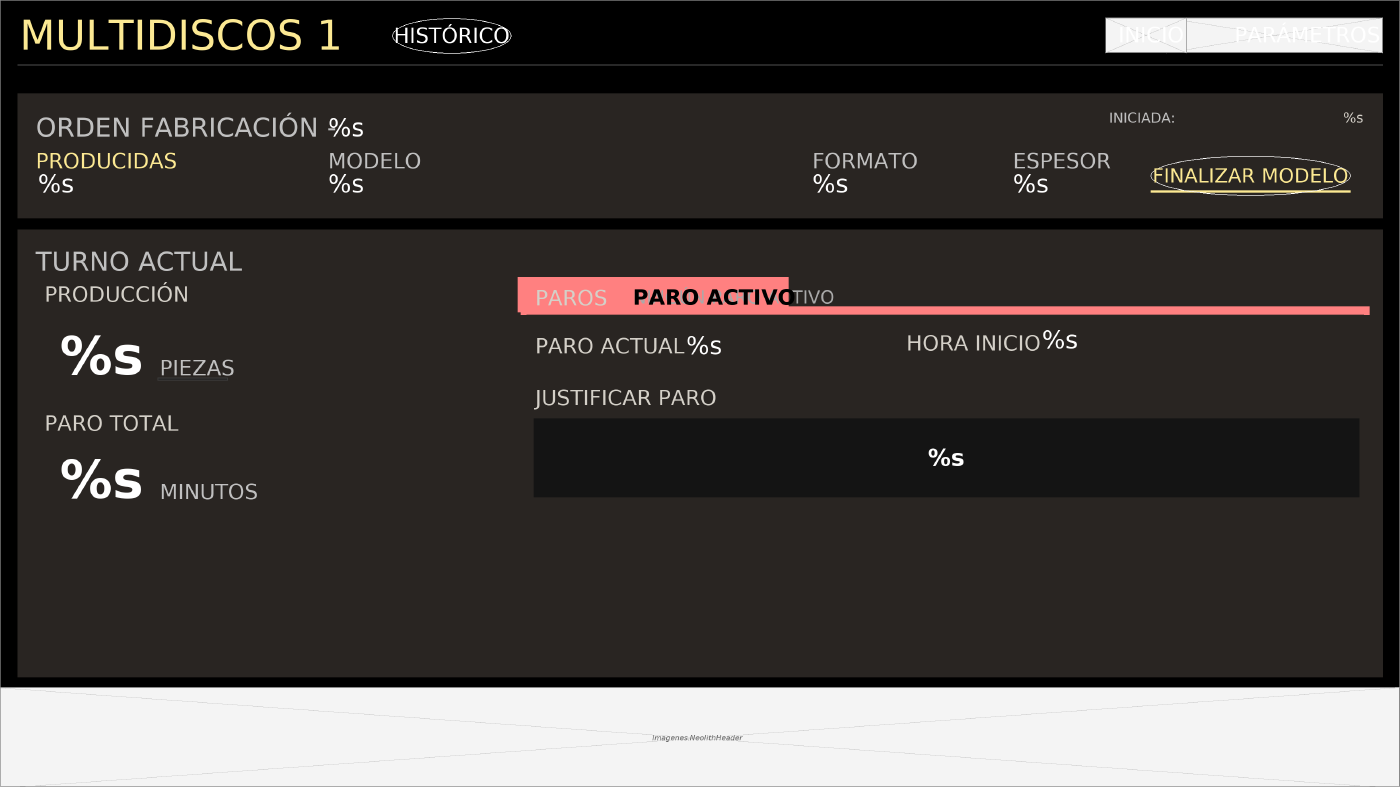
VISUALIZATION Home_Multidis1  // 1920x1080
    Ellipse (1559,1109 456x77), "Fin de producción del modelo"
        OnMouseClick: OpenDialog Dialog=V_Emerg_Fin_Prod_Md1, OpenModal=True, OpenCentered=True
    Rectangle (2270,679 183x30), "%s", text variable: FuncParoNodoMultidiscos.Funci_Multidiscos1.H_InParo_Ftc, invisible if: FuncParoNodoMultidiscos.Funci_Multidiscos1.M_SinParo_Ftc
    Label (2034,678 239x30), "Hora Inicio del paro", invisible if: FuncParoNodoMultidiscos.Funci_Multidiscos1.M_SinParo_Ftc
    Rectangle (2270,737 192x30), "%s", text variable: FuncParoNodoMultidiscos.Funci_Multidiscos1.Min_Parado_Ftc, invisible if: FuncParoNodoMultidiscos.Funci_Multidiscos1.M_SinParo_Ftc
    Label (2069,737 204x30), "Minutos Parado", invisible if: FuncParoNodoMultidiscos.Funci_Multidiscos1.M_SinParo_Ftc
    Label (2029,792 244x30), "Tiempo entre Piezas"
    Label (2018,828 255x62), "Tiempo entre Piezas Anterior"
    Rectangle (2532,486 183x123), "%s", text variable: FuncParoNodoMultidiscos.Funci_Multidiscos1.Cont_Piezas_Ftc
    Rectangle (2270,792 192x30), "%s", text variable: FuncParoNodoMultidiscos.Funci_Multidiscos1.t_Entre_Piez_Ftc
    Rectangle (2270,844 192x30), "%s", text variable: FuncParoNodoMultidiscos.Funci_Multidiscos1.t_Entr_Piez_Ante_Ftc
    Label (2029,582 326x30), "En producción todo OK", invisible if: FuncParoNodoMultidiscos.Funci_Multidiscos1.MParo_Ftc
    Label (2047,507 235x59), "Línea en paro", invisible if: FuncParoNodoMultidiscos.Funci_Multidiscos1.M_SinParo_Ftc
    Label (2424,368 354x119), "Número de losas"
    Rectangle (234,1309 1380x154), "%s", text variable: FuncParoNodoMultidiscos.Funci_Multidiscos1.S_Justi_Paro_Ftc, invisible if: FuncParoNodoMultidiscos.Funci_Multidiscos1.M_SinParo_Ftc
        OnMouseDown: write the text variable via Edit
    Label (25,1090 1381x106), "JUSTIFICAR EL PARO ACTUAL", invisible if: FuncParoNodoMultidiscos.Funci_Multidiscos1.M_SinParo_Ftc
    Image (893,-598 250x250), invisible if: FuncParoNodoMultidiscos.Funci_Multidiscos1.M_SinParo_Ftc, image: ImagePool.Exclamación
    Rectangle (24,88 1872x2)
    Label (24,16 514x64), "MULTIDISCOS 1"
    Image (1600,24 296x48), "PARÁMETROS"
        OnMouseClick: change screen: Ajustes_CorteH4
    Image (1516,24 111x48), "INICIO"
        OnMouseClick: change screen: Home_Sel_Maq
    Ellipse (538,25 163x48), "HISTÓRICO"
        OnMouseClick: change screen: HistTablaTablas_Ch4
    Rectangle (24,128 1872x171)
    Label (46,148 390x54), "ORDEN FABRICACIÓN -"
    Rectangle (1573,147 300x30), "%s", text variable: FuncParoNodoMultidiscos.sFechaInicModeloTab_MD1
    Label (1518,147 99x30), "INICIADA:"
    Rectangle (447,232 671x40), "%s", text variable: FuncParoNodoMultidiscos.sModeloActualTabla_MD1
    Rectangle (1386,232 120x40), "%s", text variable: FuncParoNodoMultidiscos.sEspesorActualTabla_MD1
    Rectangle (1111,232 321x40), "%s", text variable: FuncParoNodoMultidiscos.sFormatoActualTabla_MD1
    Label (447,203 487x36), "MODELO"
    Label (1111,203 156x36), "FORMATO"
    Label (1386,203 156x36), "ESPESOR"
    Rectangle (447,155 321x40), "%s", text variable: FuncParoNodoCorteH4Remote1.sFormatoActualTabla
    Label (46,203 199x36), "PRODUCIDAS"
    Rectangle (49,232 248x40), "%s", text variable: FuncParoNodoCorteH4Remote1.sEspesorActualTabla
    Group (1578,214 274x54)
        Rectangle (0,47 274x3)
        Ellipse (0,0 274x54), "FINALIZAR MODELO"
            OnMouseClick: OpenDialog Dialog=V_Emerg_Fin_Prod_Md1, OpenModal=True, OpenCentered=True
    Rectangle (24,315 1872x614)
    Rectangle (1426,451 401x30), "%s", text variable: FuncParoNodoMultidiscos.Funci_Multidiscos1.H_InParo_Ftc, invisible if: FuncParoNodoMultidiscos.Funci_Multidiscos1.M_SinParo_Ftc
    Rectangle (938,459 192x30), "%s", text variable: FuncParoNodoMultidiscos.Funci_Multidiscos1.Min_Parado_Ftc, invisible if: FuncParoNodoMultidiscos.Funci_Multidiscos1.M_SinParo_Ftc
    Rectangle (732,574 1132x108), "%s", text variable: FuncParoNodoMultidiscos.Funci_Multidiscos1.S_Justi_Paro_Ftc, invisible if: FuncParoNodoMultidiscos.Funci_Multidiscos1.M_SinParo_Ftc
        OnMouseDown: write the text variable via Edit
    Label (46,332 390x54), "TURNO ACTUAL"
    Label (58,386 199x36), "PRODUCCIÓN"
    Label (731,457 261x36), "PARO ACTUAL", invisible if: FuncParoNodoMultidiscos.Funci_Multidiscos1.M_SinParo_Ftc
    Label (1240,453 261x36), "HORA INICIO", invisible if: FuncParoNodoMultidiscos.Funci_Multidiscos1.M_SinParo_Ftc
    Rectangle (79,444 183x88), "%s", text variable: FuncParoNodoMultidiscos.Funci_Multidiscos1.Cont_Piezas_Ftc
    Label (216,487 106x36), "PIEZAS"
    Rectangle (216,518 96x4), colour toggle: FuncParoNodoMultidiscos.Funci_Multidiscos1.Fotocelula
    Label (731,528 261x36), "JUSTIFICAR PARO", invisible if: FuncParoNodoMultidiscos.Funci_Multidiscos1.M_SinParo_Ftc
    Group (710,380 1168x48), invisible if: FuncParoNodoMultidiscos.Funci_Multidiscos1.M_SinParo_Ftc
        Rectangle (4,44 1164x4)
        Rectangle (0,0 371x48)
        Label (21,11 199x36), "PAROS"
        Label (155,13 326x30), "NINGÚN PARO ACTIVO", invisible if: FuncParoNodoCorteH4Remote1.Funci_CortHum4.MParo_Ftc
        Label (155,13 235x30), "PARO ACTIVO", invisible if: FuncParoNodoCorteH4Remote1.Funci_CortHum4.M_SinParo_Ftc
    Label (58,563 261x36), "PARO TOTAL"
    Rectangle (79,614 183x88), "%s", text variable: FuncParoNodoCorteH4Remote1.Funci_CortHum4.Cont_Piezas_Ftc
    Label (216,657 142x36), "MINUTOS"
    Image (-7,943 1927x139), image: Imagenes.NeolithHeader
END_VISUALIZATION

